C07308=1230.127,396.275,-78.801,-175.693,7.707,148.228
C07309=1230.123,396.522,-78.835,-175.692,7.710,148.228
C07310=1230.118,396.770,-78.868,-175.691,7.712,148.229
C07311=1230.115,397.018,-78.903,-175.691,7.714,148.229
C07312=1230.110,397.266,-78.936,-175.690,7.717,148.229
C07313=1230.106,397.513,-78.970,-175.689,7.719,148.230
C07314=1230.102,397.760,-79.004,-175.688,7.722,148.230
C07315=1230.098,398.009,-79.038,-175.688,7.724,148.231
C07316=1230.094,398.256,-79.072,-175.686,7.727,148.231
C07317=1230.090,398.503,-79.106,-175.686,7.729,148.232
C07318=1230.086,398.751,-79.141,-175.685,7.731,148.232
C07319=1230.082,398.999,-79.174,-175.684,7.734,148.232
C07320=1230.078,399.246,-79.208,-175.684,7.736,148.233
C07321=1230.073,399.494,-79.243,-175.683,7.739,148.233
C07322=1230.070,399.742,-79.276,-175.682,7.741,148.234
C07323=1230.065,399.989,-79.311,-175.681,7.743,148.234
C07324=1230.061,400.237,-79.345,-175.681,7.746,148.235
C07325=1230.057,400.485,-79.379,-175.680,7.748,148.235
C07326=1230.053,400.732,-79.413,-175.679,7.750,148.235
C07327=1230.049,400.980,-79.447,-175.678,7.753,148.236
C07328=1230.045,401.228,-79.481,-175.678,7.755,148.236
C07329=1230.041,401.475,-79.516,-175.677,7.758,148.237
C07330=1230.037,401.723,-79.549,-175.676,7.760,148.237
C07331=1230.033,401.971,-79.584,-175.676,7.762,148.237
C07332=1230.029,402.218,-79.618,-175.674,7.764,148.238
C07333=1230.024,402.465,-79.652,-175.674,7.767,148.238
C07334=1230.021,402.713,-79.686,-175.674,7.769,148.239
C07335=1230.016,402.961,-79.720,-175.672,7.772,148.239
C07336=1230.012,403.208,-79.754,-175.672,7.773,148.239
C07337=1230.008,403.456,-79.789,-175.672,7.776,148.240
C07338=1230.005,403.704,-79.823,-175.671,7.778,148.240
C07339=1230.000,403.951,-79.857,-175.670,7.781,148.241
C07340=1229.997,404.199,-79.891,-175.669,7.783,148.241
C07341=1229.992,404.446,-79.926,-175.669,7.785,148.241
C07342=1229.987,404.694,-79.960,-175.668,7.788,148.242
C07343=1229.984,404.942,-79.994,-175.667,7.790,148.242
C07344=1229.979,405.190,-80.028,-175.667,7.792,148.243
C07345=1229.976,405.437,-80.062,-175.666,7.795,148.243
C07346=1229.972,405.685,-80.097,-175.665,7.797,148.243
C07347=1229.968,405.932,-80.131,-175.665,7.799,148.244
C07348=1229.963,406.179,-80.165,-175.664,7.801,148.244
C07349=1229.960,406.427,-80.200,-175.663,7.804,148.245
C07350=1229.955,406.675,-80.233,-175.663,7.806,148.245
C07351=1229.951,406.923,-80.268,-175.662,7.808,148.245
C07352=1229.947,407.170,-80.302,-175.661,7.810,148.246
C07353=1229.943,407.418,-80.337,-175.661,7.813,148.246
C07354=1229.940,407.666,-80.371,-175.660,7.815,148.247
C07355=1229.935,407.913,-80.405,-175.659,7.817,148.247
C07356=1229.930,408.160,-80.440,-175.659,7.819,148.247
C07357=1229.927,408.408,-80.474,-175.658,7.822,148.248
C07358=1229.923,408.656,-80.508,-175.658,7.824,148.248
C07359=1229.919,408.904,-80.543,-175.657,7.826,148.249
C07360=1229.915,409.151,-80.577,-175.656,7.828,148.249
C07361=1229.910,409.398,-80.612,-175.656,7.831,148.250
C07362=1229.907,409.646,-80.646,-175.655,7.833,148.250
C07363=1229.902,409.894,-80.680,-175.654,7.835,148.250
C07364=1229.898,410.142,-80.715,-175.654,7.837,148.251
C07365=1229.895,410.389,-80.749,-175.653,7.839,148.251
C07366=1229.890,410.636,-80.783,-175.652,7.842,148.252
C07367=1229.886,410.884,-80.818,-175.652,7.844,148.252
C07368=1229.882,411.131,-80.852,-175.651,7.846,148.252
C07369=1229.878,411.380,-80.887,-175.651,7.848,148.253
C07370=1229.874,411.627,-80.921,-175.650,7.850,148.253
C07371=1229.870,411.874,-80.955,-175.650,7.852,148.254
C07372=1229.866,412.122,-80.990,-175.648,7.855,148.254
C07373=1229.861,412.370,-81.025,-175.648,7.857,148.254
C07374=1229.858,412.617,-81.059,-175.648,7.859,148.255
C07375=1229.854,412.865,-81.093,-175.647,7.861,148.255
C07376=1229.849,413.112,-81.128,-175.646,7.863,148.255
C07377=1229.846,413.360,-81.162,-175.646,7.865,148.256
C07378=1229.841,413.607,-81.196,-175.645,7.868,148.256
C07379=1229.837,413.856,-81.231,-175.644,7.870,148.257
C07380=1229.834,414.102,-81.266,-175.644,7.872,148.257
C07381=1229.830,414.350,-81.301,-175.644,7.875,148.258
C07382=1229.825,414.598,-81.335,-175.643,7.876,148.258
C07383=1229.822,414.845,-81.369,-175.642,7.878,148.258
C07384=1229.817,415.093,-81.404,-175.642,7.880,148.259
C07385=1229.813,415.340,-81.438,-175.641,7.884,148.259
C07386=1229.809,415.588,-81.473,-175.640,7.886,148.260
C07387=1229.803,415.965,-81.525,-175.640,7.889,148.260
C07388=1229.797,416.341,-81.578,-175.639,7.892,148.261
C07389=1229.791,416.718,-81.631,-175.638,7.895,148.261
C07390=1229.786,417.095,-81.684,-175.636,7.899,148.262
C07391=1229.363,417.096,-81.716,-175.640,7.909,148.266
C07392=1229.368,416.716,-81.663,-175.641,7.905,148.265
C07393=1229.374,416.336,-81.610,-175.642,7.902,148.264
C07394=1229.381,415.957,-81.557,-175.643,7.899,148.264
C07395=1229.387,415.578,-81.504,-175.643,7.896,148.263
C07396=1229.391,415.330,-81.470,-175.645,7.893,148.263
C07397=1229.395,415.082,-81.435,-175.645,7.891,148.262
C07398=1229.399,414.835,-81.401,-175.646,7.889,148.262
C07399=1229.403,414.587,-81.366,-175.646,7.887,148.262
C07400=1229.408,414.340,-81.332,-175.647,7.885,148.261
C07401=1229.411,414.092,-81.297,-175.647,7.883,148.261
C07402=1229.415,413.845,-81.262,-175.648,7.881,148.261
C07403=1229.419,413.597,-81.227,-175.648,7.879,148.260
C07404=1229.424,413.349,-81.193,-175.649,7.876,148.260
C07405=1229.428,413.102,-81.159,-175.650,7.874,148.259
C07406=1229.432,412.854,-81.124,-175.651,7.872,148.259
C07407=1229.436,412.607,-81.090,-175.651,7.870,148.258
C07408=1229.439,412.359,-81.056,-175.651,7.868,148.258
C07409=1229.444,412.112,-81.021,-175.652,7.866,148.258
C07410=1229.448,411.863,-80.986,-175.653,7.862,148.257
C07411=1229.452,411.616,-80.952,-175.653,7.861,148.257
C07412=1229.456,411.369,-80.918,-175.654,7.859,148.256
C07413=1229.460,411.121,-80.883,-175.655,7.857,148.256
C07414=1229.464,410.874,-80.849,-175.655,7.854,148.256
C07415=1229.468,410.626,-80.814,-175.656,7.851,148.255
C07416=1229.473,410.378,-80.780,-175.657,7.849,148.255
C07417=1229.477,410.131,-80.746,-175.657,7.847,148.254
C07418=1229.480,409.883,-80.711,-175.657,7.845,148.254
C07419=1229.485,409.635,-80.677,-175.658,7.843,148.254
C07420=1229.488,409.388,-80.643,-175.659,7.840,148.253
C07421=1229.493,409.140,-80.608,-175.660,7.838,148.253
C07422=1229.497,408.893,-80.574,-175.660,7.836,148.252
C07423=1229.501,408.645,-80.539,-175.661,7.834,148.252
C07424=1229.505,408.398,-80.505,-175.661,7.832,148.252
C07425=1229.508,408.150,-80.471,-175.662,7.829,148.251
C07426=1229.513,407.902,-80.436,-175.663,7.827,148.251
C07427=1229.518,407.655,-80.402,-175.663,7.825,148.250
C07428=1229.521,407.407,-80.367,-175.664,7.823,148.250
C07429=1229.525,407.160,-80.333,-175.665,7.820,148.249
C07430=1229.529,406.913,-80.299,-175.665,7.818,148.249
C07431=1229.533,406.665,-80.264,-175.666,7.816,148.249
C07432=1229.538,406.417,-80.230,-175.666,7.814,148.248
C07433=1229.541,406.169,-80.196,-175.667,7.811,148.248
C07434=1229.546,405.922,-80.161,-175.668,7.809,148.247
C07435=1229.550,405.674,-80.128,-175.668,7.807,148.247
C07436=1229.554,405.426,-80.093,-175.670,7.804,148.247
C07437=1229.558,405.179,-80.059,-175.670,7.802,148.246
C07438=1229.562,404.931,-80.025,-175.670,7.800,148.246
C07439=1229.566,404.683,-79.990,-175.671,7.798,148.245
C07440=1229.570,404.436,-79.956,-175.672,7.795,148.245
C07441=1229.574,404.189,-79.922,-175.672,7.793,148.244
C07442=1229.578,403.941,-79.887,-175.673,7.791,148.244
C07443=1229.583,403.693,-79.854,-175.674,7.788,148.244
C07444=1229.586,403.446,-79.820,-175.675,7.786,148.243
C07445=1229.590,403.198,-79.785,-175.675,7.784,148.243
C07446=1229.594,402.951,-79.751,-175.676,7.781,148.242
C07447=1229.598,402.703,-79.716,-175.677,7.779,148.242
C07448=1229.602,402.455,-79.682,-175.677,7.777,148.242
C07449=1229.607,402.207,-79.649,-175.678,7.774,148.241
C07450=1229.610,401.960,-79.614,-175.679,7.772,148.241
C07451=1229.615,401.712,-79.580,-175.679,7.770,148.240
C07452=1229.619,401.465,-79.545,-175.681,7.767,148.240
C07453=1229.623,401.218,-79.512,-175.681,7.765,148.240
C07454=1229.627,400.969,-79.477,-175.681,7.763,148.239
C07455=1229.631,400.722,-79.444,-175.683,7.760,148.239
C07456=1229.636,400.474,-79.409,-175.683,7.758,148.238
C07457=1229.639,400.227,-79.375,-175.684,7.756,148.238
C07458=1229.644,399.978,-79.341,-175.684,7.753,148.238
C07459=1229.648,399.731,-79.307,-175.685,7.751,148.237
C07460=1229.651,399.484,-79.273,-175.686,7.748,148.237
C07461=1229.655,399.236,-79.239,-175.687,7.746,148.236
C07462=1229.660,398.988,-79.205,-175.687,7.744,148.236
C07463=1229.664,398.740,-79.171,-175.688,7.741,148.235
C07464=1229.667,398.493,-79.137,-175.689,7.739,148.235
C07465=1229.672,398.245,-79.103,-175.690,7.736,148.235
C07466=1229.676,397.998,-79.069,-175.691,7.734,148.234
C07467=1229.680,397.750,-79.034,-175.691,7.732,148.234
C07468=1229.684,397.502,-79.001,-175.692,7.729,148.233
C07469=1229.689,397.255,-78.967,-175.693,7.727,148.233
C07470=1229.692,397.007,-78.932,-175.694,7.724,148.233
C07471=1229.696,396.759,-78.899,-175.694,7.722,148.232
C07472=1229.701,396.512,-78.865,-175.695,7.719,148.232
C07473=1229.705,396.265,-78.831,-175.696,7.717,148.231
C07474=1229.709,396.016,-78.797,-175.696,7.715,148.231
C07475=1229.713,395.769,-78.763,-175.698,7.713,148.231
C07476=1229.717,395.521,-78.728,-175.698,7.711,148.230
C07477=1229.721,395.274,-78.695,-175.699,7.707,148.230
C07478=1229.725,395.026,-78.661,-175.700,7.705,148.229
C07479=1229.729,394.778,-78.627,-175.701,7.703,148.229
C07480=1229.733,394.531,-78.593,-175.701,7.701,148.229
C07481=1229.738,394.283,-78.559,-175.702,7.698,148.228
C07482=1229.741,394.035,-78.525,-175.703,7.696,148.228
C07483=1229.745,393.788,-78.492,-175.704,7.693,148.227
C07484=1229.750,393.506,-78.453,-175.705,7.690,148.227
C07485=1229.755,393.225,-78.414,-175.706,7.688,148.227
C07486=1229.759,392.944,-78.375,-175.707,7.685,148.226
C07487=1229.764,392.662,-78.338,-175.708,7.682,148.226
C07488=1229.768,392.415,-78.304,-175.709,7.679,148.225
C07489=1229.773,392.167,-78.270,-175.709,7.677,148.225
C07490=1229.776,391.919,-78.236,-175.710,7.674,148.224
C07491=1229.780,391.672,-78.203,-175.711,7.672,148.224
C07492=1229.785,391.424,-78.168,-175.712,7.670,148.224
C07493=1229.789,391.176,-78.135,-175.712,7.667,148.223
C07494=1229.792,390.929,-78.101,-175.714,7.664,148.223
C07495=1229.797,390.681,-78.067,-175.715,7.662,148.222
C07496=1229.801,390.434,-78.033,-175.715,7.660,148.222
C07497=1229.805,390.186,-78.000,-175.717,7.657,148.222
C07498=1229.809,389.938,-77.965,-175.717,7.655,148.221
C07499=1229.813,389.690,-77.932,-175.718,7.652,148.221
C07500=1229.817,389.443,-77.898,-175.719,7.650,148.220
C07501=1229.821,389.195,-77.865,-175.720,7.647,148.220
C07502=1229.826,388.947,-77.831,-175.721,7.644,148.220
C07503=1229.829,388.699,-77.797,-175.722,7.642,148.219
C07504=1229.834,388.452,-77.764,-175.723,7.639,148.219
C07505=1229.838,388.204,-77.729,-175.723,7.637,148.218
C07506=1229.842,387.956,-77.696,-175.724,7.634,148.218
C07507=1229.846,387.709,-77.662,-175.726,7.632,148.218
C07508=1229.850,387.461,-77.629,-175.726,7.630,148.217
C07509=1229.855,387.213,-77.595,-175.727,7.627,148.217
C07510=1229.858,386.966,-77.561,-175.729,7.624,148.216
C07511=1229.862,386.718,-77.528,-175.729,7.622,148.216
C07512=1229.867,386.470,-77.495,-175.730,7.619,148.216
C07513=1229.871,386.223,-77.460,-175.732,7.616,148.215
C07514=1229.875,385.974,-77.427,-175.732,7.614,148.215
C07515=1229.879,385.727,-77.394,-175.733,7.612,148.215
C07516=1229.883,385.480,-77.360,-175.734,7.609,148.214
C07517=1229.887,385.232,-77.327,-175.735,7.607,148.214
C07518=1229.892,384.984,-77.293,-175.736,7.604,148.213
C07519=1229.896,384.737,-77.259,-175.737,7.601,148.213
C07520=1229.900,384.489,-77.226,-175.738,7.599,148.213
C07521=1229.903,384.241,-77.192,-175.739,7.596,148.212
C07522=1229.908,383.993,-77.158,-175.740,7.594,148.212
C07523=1229.912,383.745,-77.125,-175.741,7.592,148.212
C07524=1229.916,383.498,-77.092,-175.742,7.589,148.211
C07525=1229.920,383.250,-77.059,-175.743,7.586,148.211
C07526=1229.924,383.003,-77.025,-175.744,7.584,148.210
C07527=1229.928,382.755,-76.992,-175.745,7.581,148.210
C07528=1229.932,382.506,-76.957,-175.746,7.578,148.210
C07529=1229.937,382.259,-76.924,-175.747,7.575,148.209
C07530=1229.940,382.012,-76.890,-175.748,7.573,148.209
C07531=1229.945,381.764,-76.857,-175.749,7.571,148.208
C07532=1229.949,381.516,-76.824,-175.750,7.568,148.208
C07533=1229.953,381.268,-76.791,-175.752,7.565,148.208
C07534=1229.957,381.021,-76.758,-175.753,7.563,148.207
C07535=1229.962,380.773,-76.723,-175.754,7.560,148.207
C07536=1229.966,380.525,-76.690,-175.755,7.558,148.207
C07537=1229.970,380.278,-76.657,-175.756,7.555,148.206
C07538=1229.973,380.029,-76.623,-175.757,7.553,148.206
C07539=1229.978,379.782,-76.590,-175.758,7.550,148.206
C07540=1229.982,379.534,-76.557,-175.759,7.547,148.205
C07541=1229.985,379.287,-76.523,-175.760,7.544,148.205
C07542=1229.990,379.039,-76.490,-175.761,7.542,148.204
C07543=1229.994,378.791,-76.457,-175.763,7.540,148.204
C07544=1229.999,378.543,-76.423,-175.764,7.537,148.204
C07545=1230.003,378.295,-76.390,-175.765,7.534,148.203
C07546=1230.007,378.048,-76.357,-175.766,7.531,148.203
C07547=1230.011,377.800,-76.324,-175.767,7.529,148.203
C07548=1230.015,377.552,-76.291,-175.768,7.527,148.202
C07549=1230.019,377.305,-76.257,-175.769,7.524,148.202
C07550=1230.023,377.057,-76.224,-175.771,7.521,148.202
C07551=1230.028,376.809,-76.191,-175.772,7.518,148.201
C07552=1230.031,376.561,-76.158,-175.773,7.516,148.201
C07553=1230.035,376.314,-76.124,-175.774,7.513,148.200
C07554=1230.039,376.066,-76.091,-175.775,7.511,148.200
C07555=1230.043,375.818,-76.057,-175.776,7.508,148.200
C07556=1230.047,375.570,-76.024,-175.777,7.505,148.200
C07557=1230.052,375.323,-75.991,-175.779,7.503,148.199
C07558=1230.056,375.075,-75.958,-175.780,7.500,148.199
C07559=1230.060,374.827,-75.925,-175.781,7.497,148.199
C07560=1230.064,374.579,-75.892,-175.783,7.494,148.198
C07561=1230.068,374.331,-75.859,-175.784,7.492,148.198
C07562=1230.073,374.083,-75.826,-175.784,7.490,148.197
C07563=1230.077,373.836,-75.793,-175.786,7.487,148.197
C07564=1230.081,373.588,-75.760,-175.787,7.484,148.197
C07565=1230.085,373.340,-75.727,-175.788,7.481,148.196
C07566=1230.089,373.092,-75.693,-175.790,7.479,148.196
C07567=1230.093,372.845,-75.660,-175.791,7.476,148.196
C07568=1230.097,372.597,-75.627,-175.792,7.473,148.195
C07569=1230.101,372.349,-75.594,-175.793,7.470,148.195
C07570=1230.106,372.102,-75.561,-175.795,7.468,148.195
C07571=1230.110,371.854,-75.528,-175.796,7.465,148.194
C07572=1230.114,371.606,-75.494,-175.798,7.463,148.194
C07573=1230.118,371.358,-75.462,-175.799,7.460,148.194
C07574=1230.122,371.110,-75.429,-175.800,7.457,148.193
C07575=1230.126,370.863,-75.396,-175.801,7.455,148.193
C07576=1230.130,370.615,-75.363,-175.802,7.452,148.193
C07577=1230.134,370.367,-75.330,-175.804,7.450,148.193
C07578=1230.138,370.119,-75.297,-175.805,7.447,148.192
C07579=1230.143,369.871,-75.264,-175.806,7.444,148.192
C07580=1230.147,369.623,-75.231,-175.808,7.442,148.192
C07581=1230.151,369.376,-75.198,-175.809,7.439,148.191
C07582=1230.156,369.129,-75.165,-175.810,7.436,148.191
C07583=1230.160,368.881,-75.132,-175.812,7.433,148.191
C07584=1230.164,368.633,-75.100,-175.813,7.431,148.190
C07585=1230.168,368.385,-75.067,-175.815,7.428,148.190
C07586=1230.172,368.137,-75.034,-175.816,7.425,148.190
C07587=1230.176,367.890,-75.001,-175.818,7.423,148.190
C07588=1230.181,367.609,-74.964,-175.819,7.419,148.189
C07589=1230.185,367.330,-74.927,-175.820,7.416,148.189
C07590=1230.190,367.051,-74.891,-175.822,7.414,148.189
C07591=1230.195,366.771,-74.853,-175.824,7.410,148.188
C07592=1230.199,366.523,-74.820,-175.825,7.408,148.188
C07593=1230.202,366.276,-74.787,-175.826,7.405,148.188
C07594=1230.207,366.028,-74.755,-175.828,7.402,148.187
C07595=1230.211,365.780,-74.722,-175.829,7.399,148.187
C07596=1230.215,365.531,-74.689,-175.831,7.397,148.187
C07597=1230.220,365.284,-74.656,-175.832,7.394,148.186
C07598=1230.224,365.037,-74.624,-175.834,7.391,148.186
C07599=1230.228,364.789,-74.592,-175.835,7.389,148.186
C07600=1230.232,364.541,-74.558,-175.836,7.386,148.186
C07601=1230.236,364.293,-74.525,-175.838,7.384,148.185
C07602=1230.240,364.045,-74.493,-175.839,7.381,148.185
C07603=1230.244,363.797,-74.460,-175.841,7.378,148.185
C07604=1230.249,363.549,-74.428,-175.842,7.375,148.184
C07605=1230.253,363.301,-74.395,-175.844,7.373,148.184
C07606=1230.256,363.053,-74.363,-175.845,7.370,148.184
C07607=1230.261,362.806,-74.330,-175.847,7.367,148.184
C07608=1230.265,362.559,-74.297,-175.849,7.364,148.183
C07609=1230.269,362.311,-74.265,-175.850,7.361,148.183
C07610=1230.273,362.063,-74.232,-175.851,7.359,148.183
C07611=1230.278,361.814,-74.199,-175.853,7.356,148.183
C07612=1230.281,361.567,-74.167,-175.854,7.353,148.182
C07613=1230.285,361.319,-74.134,-175.856,7.351,148.182
C07614=1230.290,361.072,-74.102,-175.857,7.348,148.182
C07615=1230.294,360.824,-74.070,-175.859,7.346,148.181
C07616=1230.298,360.575,-74.037,-175.860,7.343,148.181
C07617=1230.302,360.328,-74.004,-175.862,7.340,148.181
C07618=1230.306,360.080,-73.972,-175.864,7.337,148.181
C07619=1230.310,359.832,-73.939,-175.865,7.334,148.180
C07620=1230.315,359.584,-73.907,-175.867,7.332,148.180
C07621=1230.319,359.337,-73.875,-175.868,7.329,148.180
C07622=1230.323,359.088,-73.842,-175.870,7.327,148.180
C07623=1230.328,358.840,-73.810,-175.871,7.324,148.179
C07624=1230.331,358.593,-73.777,-175.873,7.321,148.179
C07625=1230.336,358.345,-73.745,-175.874,7.319,148.179
C07626=1230.339,358.098,-73.712,-175.877,7.315,148.179
C07627=1230.344,357.849,-73.680,-175.878,7.313,148.178
C07628=1230.348,357.601,-73.648,-175.879,7.310,148.178
C07629=1230.352,357.353,-73.615,-175.881,7.308,148.178
C07630=1230.357,357.106,-73.583,-175.883,7.305,148.178
C07631=1230.361,356.858,-73.551,-175.884,7.302,148.178
C07632=1230.365,356.609,-73.519,-175.885,7.300,148.177
C07633=1230.368,356.362,-73.486,-175.887,7.297,148.177
C07634=1230.373,356.114,-73.454,-175.889,7.294,148.177
C07635=1230.378,355.866,-73.422,-175.891,7.291,148.177
C07636=1230.381,355.619,-73.389,-175.892,7.289,148.177
C07637=1230.386,355.370,-73.357,-175.894,7.286,148.176
C07638=1230.390,355.123,-73.325,-175.895,7.283,148.176
C07639=1230.394,354.875,-73.293,-175.897,7.281,148.176
C07640=1230.398,354.627,-73.260,-175.899,7.277,148.176
C07641=1230.402,354.379,-73.228,-175.901,7.275,148.175
C07642=1230.407,354.131,-73.196,-175.902,7.272,148.175
C07643=1230.411,353.883,-73.164,-175.904,7.270,148.175
C07644=1230.415,353.635,-73.132,-175.906,7.267,148.175
C07645=1230.419,353.387,-73.099,-175.907,7.265,148.175
C07646=1230.423,353.140,-73.067,-175.909,7.261,148.174
C07647=1230.428,352.892,-73.035,-175.911,7.259,148.174
C07648=1230.431,352.644,-73.003,-175.912,7.256,148.174
C07649=1230.436,352.396,-72.971,-175.914,7.253,148.174
C07650=1230.440,352.148,-72.939,-175.915,7.251,148.173
C07651=1230.445,351.900,-72.907,-175.917,7.248,148.173
C07652=1230.448,351.651,-72.875,-175.919,7.245,148.173
C07653=1230.452,351.405,-72.843,-175.921,7.243,148.173
C07654=1230.457,351.156,-72.810,-175.922,7.240,148.173
C07655=1230.460,350.908,-72.778,-175.924,7.237,148.172
C07656=1230.465,350.661,-72.746,-175.926,7.235,148.172
C07657=1230.469,350.413,-72.714,-175.927,7.232,148.172
C07658=1230.473,350.165,-72.683,-175.929,7.229,148.172
C07659=1230.478,349.917,-72.650,-175.931,7.226,148.172
C07660=1230.482,349.669,-72.619,-175.933,7.224,148.172
C07661=1230.486,349.421,-72.586,-175.934,7.221,148.171
C07662=1230.490,349.173,-72.555,-175.936,7.219,148.171
C07663=1230.494,348.925,-72.523,-175.938,7.216,148.171
C07664=1230.499,348.677,-72.490,-175.940,7.213,148.171
C07665=1230.503,348.430,-72.459,-175.941,7.210,148.171
C07666=1230.507,348.182,-72.427,-175.943,7.208,148.171
C07667=1230.511,347.933,-72.395,-175.945,7.206,148.170
C07668=1230.515,347.686,-72.363,-175.947,7.202,148.170
C07669=1230.519,347.438,-72.331,-175.949,7.200,148.170
C07670=1230.524,347.190,-72.300,-175.951,7.197,148.170
C07671=1230.528,346.941,-72.268,-175.952,7.195,148.170
C07672=1230.532,346.693,-72.236,-175.954,7.191,148.169
C07673=1230.537,346.446,-72.204,-175.956,7.189,148.169
C07674=1230.541,346.198,-72.172,-175.958,7.186,148.169
C07675=1230.545,345.950,-72.141,-175.959,7.184,148.169
C07676=1230.549,345.702,-72.108,-175.961,7.182,148.169
C07677=1230.553,345.454,-72.077,-175.963,7.178,148.169
C07678=1230.558,345.206,-72.046,-175.965,7.176,148.168
C07679=1230.561,344.958,-72.014,-175.967,7.173,148.168
C07680=1230.566,344.710,-71.982,-175.968,7.171,148.168
C07681=1230.570,344.462,-71.950,-175.970,7.167,148.168
C07682=1230.574,344.214,-71.918,-175.973,7.165,148.168
C07683=1230.578,343.966,-71.887,-175.974,7.162,148.168
C07684=1230.583,343.718,-71.855,-175.976,7.160,148.168
C07685=1230.587,343.471,-71.824,-175.977,7.157,148.167
C07686=1230.591,343.223,-71.792,-175.980,7.154,148.167
C07687=1230.595,342.975,-71.761,-175.982,7.152,148.167
C07688=1230.600,342.726,-71.728,-175.983,7.149,148.167
C07689=1230.604,342.478,-71.697,-175.985,7.147,148.167
C07690=1230.608,342.231,-71.665,-175.987,7.143,148.167
C07691=1230.612,341.982,-71.634,-175.989,7.141,148.167
C07692=1230.617,341.705,-71.599,-175.991,7.139,148.166
C07693=1230.621,341.428,-71.563,-175.993,7.135,148.166
C07694=1230.626,341.149,-71.528,-175.995,7.132,148.166
C07695=1230.631,340.873,-71.492,-175.997,7.130,148.166
C07696=1230.635,340.624,-71.461,-175.999,7.126,148.166
C07697=1230.640,340.377,-71.430,-176.001,7.124,148.166
C07698=1230.643,340.129,-71.398,-176.003,7.121,148.166
C07699=1230.648,339.881,-71.367,-176.005,7.119,148.165
C07700=1230.652,339.633,-71.335,-176.007,7.116,148.165
C07701=1230.656,339.385,-71.305,-176.009,7.113,148.165
C07702=1230.661,339.136,-71.272,-176.011,7.111,148.165
C07703=1230.665,338.889,-71.241,-176.012,7.108,148.165
C07704=1230.669,338.640,-71.210,-176.014,7.105,148.165
C07705=1230.673,338.393,-71.178,-176.017,7.103,148.165
C07706=1230.677,338.144,-71.147,-176.018,7.100,148.164
C07707=1230.682,337.897,-71.115,-176.020,7.098,148.164
C07708=1230.686,337.648,-71.084,-176.022,7.095,148.164
C07709=1230.690,337.401,-71.053,-176.024,7.092,148.164
C07710=1230.694,337.152,-71.022,-176.026,7.090,148.164
C07711=1230.698,336.905,-70.990,-176.028,7.087,148.164
C07712=1230.702,336.656,-70.959,-176.030,7.084,148.164
C07713=1230.707,336.409,-70.928,-176.032,7.082,148.164
C07714=1230.711,336.160,-70.897,-176.034,7.079,148.164
C07715=1230.715,335.913,-70.865,-176.036,7.077,148.164
C07716=1230.719,335.664,-70.834,-176.038,7.074,148.163
C07717=1230.724,335.416,-70.803,-176.040,7.071,148.163
C07718=1230.728,335.169,-70.772,-176.042,7.069,148.163
C07719=1230.732,334.920,-70.741,-176.043,7.066,148.163
C07720=1230.736,334.673,-70.709,-176.046,7.063,148.163
C07721=1230.740,334.424,-70.678,-176.048,7.061,148.163
C07722=1230.745,334.176,-70.647,-176.049,7.058,148.163
C07723=1230.749,333.928,-70.615,-176.051,7.056,148.163
C07724=1230.753,333.680,-70.585,-176.053,7.053,148.163
C07725=1230.758,333.432,-70.554,-176.056,7.050,148.163
C07726=1230.762,333.184,-70.522,-176.057,7.048,148.162
C07727=1230.766,332.936,-70.491,-176.060,7.045,148.162
C07728=1230.770,332.688,-70.460,-176.061,7.042,148.162
C07729=1230.774,332.440,-70.429,-176.064,7.040,148.162
C07730=1230.779,332.193,-70.398,-176.065,7.037,148.162
C07731=1230.783,331.944,-70.367,-176.068,7.034,148.162
C07732=1230.787,331.696,-70.337,-176.069,7.032,148.162
C07733=1230.791,331.449,-70.305,-176.072,7.030,148.162
C07734=1230.795,331.200,-70.274,-176.073,7.027,148.162
C07735=1230.800,330.952,-70.243,-176.076,7.024,148.162
C07736=1230.804,330.704,-70.212,-176.077,7.021,148.162
C07737=1230.809,330.456,-70.181,-176.080,7.019,148.162
C07738=1230.813,330.208,-70.150,-176.082,7.016,148.161
C07739=1230.817,329.960,-70.119,-176.084,7.014,148.161
C07740=1230.821,329.712,-70.088,-176.086,7.011,148.161
C07741=1230.825,329.464,-70.058,-176.088,7.009,148.161
C07742=1230.829,329.215,-70.027,-176.090,7.006,148.161
C07743=1230.834,328.967,-69.996,-176.092,7.003,148.161
C07744=1230.838,328.720,-69.964,-176.094,7.001,148.161
C07745=1230.842,328.472,-69.934,-176.095,6.999,148.161
C07746=1230.846,328.224,-69.903,-176.098,6.995,148.161
C07747=1230.851,327.976,-69.872,-176.100,6.993,148.161
C07748=1230.855,327.727,-69.841,-176.102,6.991,148.161
C07749=1230.859,327.479,-69.810,-176.104,6.988,148.161
C07750=1230.863,327.232,-69.780,-176.106,6.985,148.161
C07751=1230.868,326.984,-69.749,-176.108,6.983,148.161
C07752=1230.872,326.735,-69.718,-176.110,6.981,148.161
C07753=1230.877,326.487,-69.688,-176.112,6.977,148.160
C07754=1230.880,326.239,-69.657,-176.115,6.975,148.161
C07755=1230.884,325.991,-69.626,-176.117,6.973,148.161
C07756=1230.889,325.743,-69.596,-176.118,6.970,148.160
C07757=1230.894,325.495,-69.565,-176.121,6.967,148.160
C07758=1230.898,325.247,-69.535,-176.123,6.965,148.160
C07759=1230.902,324.998,-69.503,-176.125,6.962,148.160
C07760=1230.906,324.750,-69.473,-176.127,6.959,148.160
C07761=1230.910,324.503,-69.443,-176.129,6.957,148.160
C07762=1230.914,324.254,-69.411,-176.131,6.955,148.160
C07763=1230.919,324.006,-69.381,-176.133,6.952,148.160
C07764=1230.923,323.759,-69.350,-176.136,6.949,148.160
C07765=1230.927,323.511,-69.320,-176.137,6.947,148.160
C07766=1230.932,323.263,-69.289,-176.140,6.945,148.160
C07767=1230.935,323.014,-69.259,-176.142,6.941,148.160
C07768=1230.940,322.766,-69.228,-176.144,6.939,148.160
C07769=1230.945,322.518,-69.198,-176.146,6.937,148.160
C07770=1230.948,322.270,-69.167,-176.148,6.935,148.160
C07771=1230.952,322.021,-69.136,-176.151,6.931,148.160
C07772=1230.956,321.774,-69.106,-176.153,6.929,148.160
C07773=1230.961,321.525,-69.076,-176.154,6.927,148.160
C07774=1230.966,321.277,-69.045,-176.156,6.924,148.160
C07775=1230.970,321.030,-69.015,-176.159,6.921,148.160
C07776=1230.974,320.781,-68.984,-176.161,6.919,148.160
C07777=1230.978,320.533,-68.954,-176.163,6.917,148.160
C07778=1230.983,320.285,-68.924,-176.165,6.914,148.160
C07779=1230.987,320.037,-68.893,-176.168,6.911,148.160
C07780=1230.991,319.789,-68.863,-176.170,6.909,148.160
C07781=1230.995,319.540,-68.832,-176.171,6.907,148.160
C07782=1230.999,319.292,-68.802,-176.174,6.904,148.160
C07783=1231.004,319.044,-68.771,-176.176,6.901,148.160
C07784=1231.008,318.797,-68.741,-176.178,6.899,148.160
C07785=1231.013,318.548,-68.711,-176.181,6.896,148.160
C07786=1231.017,318.300,-68.681,-176.182,6.893,148.160
C07787=1231.021,318.052,-68.650,-176.184,6.891,148.160
C07788=1231.025,317.803,-68.621,-176.187,6.889,148.160
C07789=1231.029,317.556,-68.590,-176.189,6.886,148.160
C07790=1231.033,317.307,-68.560,-176.191,6.884,148.160
C07791=1231.038,317.059,-68.530,-176.193,6.882,148.160
C07792=1231.042,316.812,-68.499,-176.195,6.879,148.160
C07793=1231.047,316.563,-68.469,-176.198,6.876,148.160
C07794=1231.051,316.315,-68.439,-176.200,6.874,148.160
C07795=1231.055,316.066,-68.409,-176.202,6.871,148.160
C07796=1231.060,315.791,-68.375,-176.205,6.868,148.160
C07797=1231.065,315.515,-68.342,-176.207,6.865,148.160
C07798=1231.069,315.239,-68.308,-176.209,6.863,148.160
C07799=1231.074,314.964,-68.276,-176.212,6.860,148.160
C07800=1231.078,314.716,-68.245,-176.214,6.858,148.160
C07801=1231.083,314.468,-68.215,-176.216,6.856,148.160
C07802=1231.087,314.220,-68.185,-176.219,6.853,148.160
C07803=1231.091,313.971,-68.155,-176.221,6.850,148.160
C07804=1231.095,313.723,-68.125,-176.223,6.848,148.160
C07805=1231.100,313.475,-68.095,-176.225,6.846,148.160
C07806=1231.103,313.227,-68.064,-176.227,6.842,148.160
C07807=1231.108,312.978,-68.034,-176.229,6.840,148.160
C07808=1231.113,312.730,-68.005,-176.231,6.838,148.160
C07809=1231.116,312.483,-67.975,-176.234,6.835,148.160
C07810=1231.121,312.234,-67.945,-176.236,6.833,148.160
C07811=1231.125,311.986,-67.915,-176.238,6.831,148.160
C07812=1231.129,311.738,-67.885,-176.240,6.828,148.160
C07813=1231.134,311.490,-67.855,-176.243,6.825,148.160
C07814=1231.138,311.242,-67.825,-176.245,6.823,148.160
C07815=1231.142,310.994,-67.795,-176.247,6.821,148.160
C07816=1231.147,310.745,-67.766,-176.249,6.819,148.160
C07817=1231.151,310.497,-67.735,-176.252,6.815,148.160
C07818=1231.155,310.249,-67.706,-176.254,6.813,148.160
C07819=1231.160,310.001,-67.676,-176.256,6.811,148.160
C07820=1231.164,309.752,-67.646,-176.258,6.809,148.160
C07821=1231.168,309.505,-67.616,-176.261,6.806,148.160
C07822=1231.173,309.256,-67.587,-176.263,6.804,148.160
C07823=1231.177,309.008,-67.557,-176.265,6.801,148.160
C07824=1231.182,308.759,-67.527,-176.268,6.798,148.160
C07825=1231.186,308.512,-67.497,-176.270,6.796,148.160
C07826=1231.190,308.264,-67.467,-176.272,6.794,148.160
C07827=1231.194,308.015,-67.438,-176.274,6.792,148.160
C07828=1231.198,307.767,-67.409,-176.277,6.789,148.160
C07829=1231.203,307.518,-67.379,-176.279,6.786,148.161
C07830=1231.207,307.271,-67.348,-176.281,6.784,148.161
C07831=1231.211,307.023,-67.319,-176.283,6.782,148.161
C07832=1231.215,306.774,-67.289,-176.286,6.779,148.161
C07833=1231.219,306.526,-67.260,-176.288,6.777,148.161
C07834=1231.224,306.277,-67.230,-176.290,6.774,148.161
C07835=1231.228,306.029,-67.200,-176.292,6.772,148.161
C07836=1231.233,305.781,-67.171,-176.295,6.769,148.161
C07837=1231.237,305.533,-67.142,-176.297,6.767,148.161
C07838=1231.242,305.285,-67.112,-176.299,6.765,148.161
C07839=1231.246,305.037,-67.082,-176.301,6.762,148.161
C07840=1231.250,304.789,-67.053,-176.304,6.760,148.161
C07841=1231.255,304.541,-67.023,-176.306,6.757,148.161
C07842=1231.259,304.292,-66.993,-176.308,6.755,148.161
C07843=1231.263,304.044,-66.964,-176.310,6.753,148.161
C07844=1231.267,303.796,-66.934,-176.313,6.750,148.161
C07845=1231.271,303.548,-66.905,-176.315,6.748,148.161
C07846=1231.276,303.299,-66.876,-176.317,6.745,148.161
C07847=1231.280,303.052,-66.846,-176.319,6.743,148.162
C07848=1231.284,302.803,-66.817,-176.322,6.740,148.162
C07849=1231.289,302.555,-66.788,-176.325,6.738,148.162
C07850=1231.293,302.306,-66.759,-176.327,6.736,148.162
C07851=1231.297,302.058,-66.729,-176.329,6.734,148.162
C07852=1231.302,301.810,-66.700,-176.331,6.731,148.162
C07853=1231.306,301.561,-66.670,-176.334,6.729,148.162
C07854=1231.310,301.313,-66.641,-176.336,6.726,148.162
C07855=1231.315,301.066,-66.612,-176.338,6.724,148.162
C07856=1231.319,300.817,-66.582,-176.340,6.722,148.162
C07857=1231.323,300.569,-66.553,-176.343,6.719,148.162
C07858=1231.327,300.321,-66.524,-176.345,6.717,148.162
C07859=1231.332,300.072,-66.495,-176.347,6.715,148.162
C07860=1231.336,299.824,-66.465,-176.349,6.712,148.163
C07861=1231.341,299.576,-66.436,-176.352,6.709,148.163
C07862=1231.345,299.328,-66.407,-176.355,6.707,148.163
C07863=1231.349,299.080,-66.377,-176.357,6.705,148.163
C07864=1231.354,298.831,-66.349,-176.359,6.703,148.163
C07865=1231.358,298.582,-66.319,-176.361,6.700,148.163
C07866=1231.362,298.335,-66.290,-176.364,6.698,148.163
C07867=1231.367,298.087,-66.261,-176.366,6.696,148.163
C07868=1231.371,297.838,-66.232,-176.368,6.694,148.163
C07869=1231.375,297.589,-66.202,-176.370,6.691,148.163
C07870=1231.380,297.341,-66.173,-176.373,6.688,148.163
C07871=1231.384,297.094,-66.144,-176.375,6.686,148.163
C07872=1231.389,296.845,-66.115,-176.378,6.684,148.164
C07873=1231.392,296.597,-66.086,-176.380,6.682,148.164
C07874=1231.396,296.348,-66.057,-176.382,6.679,148.164
C07875=1231.401,296.100,-66.028,-176.385,6.677,148.164
C07876=1231.406,295.852,-65.999,-176.387,6.674,148.164
C07877=1231.410,295.604,-65.970,-176.389,6.673,148.164
C07878=1231.414,295.355,-65.941,-176.391,6.670,148.164
C07879=1231.418,295.107,-65.912,-176.394,6.667,148.164
C07880=1231.423,294.859,-65.884,-176.396,6.665,148.164
C07881=1231.427,294.610,-65.854,-176.399,6.663,148.165
C07882=1231.431,294.362,-65.825,-176.401,6.661,148.165
C07883=1231.436,294.113,-65.796,-176.403,6.658,148.165
C07884=1231.441,293.866,-65.767,-176.406,6.656,148.165
C07885=1231.444,293.617,-65.739,-176.408,6.654,148.165
C07886=1231.448,293.369,-65.709,-176.410,6.652,148.165
C07887=1231.454,293.121,-65.681,-176.412,6.649,148.165
C07888=1231.458,292.872,-65.651,-176.416,6.647,148.165
C07889=1231.461,292.624,-65.623,-176.418,6.644,148.165
C07890=1231.466,292.376,-65.594,-176.420,6.642,148.165
C07891=1231.471,292.127,-65.565,-176.422,6.640,148.166
C07892=1231.475,291.879,-65.536,-176.424,6.638,148.166
C07893=1231.479,291.631,-65.508,-176.427,6.635,148.166
C07894=1231.483,291.383,-65.479,-176.429,6.633,148.166
C07895=1231.488,291.134,-65.450,-176.432,6.631,148.166
C07896=1231.492,290.886,-65.421,-176.434,6.629,148.166
C07897=1231.496,290.638,-65.393,-176.436,6.626,148.166
C07898=1231.501,290.389,-65.364,-176.439,6.624,148.167
C07899=1231.505,290.141,-65.335,-176.441,6.621,148.167
C07900=1231.511,289.867,-65.303,-176.443,6.619,148.167
C07901=1231.515,289.593,-65.272,-176.446,6.616,148.167
C07902=1231.519,289.319,-65.241,-176.449,6.614,148.167
C07903=1231.524,289.044,-65.209,-176.452,6.611,148.167
C07904=1231.529,288.797,-65.180,-176.454,6.609,148.167
C07905=1231.533,288.548,-65.152,-176.456,6.607,148.168
C07906=1231.537,288.299,-65.123,-176.459,6.605,148.168
C07907=1231.542,288.052,-65.094,-176.461,6.602,148.168
C07908=1231.546,287.803,-65.066,-176.464,6.600,148.168
C07909=1231.551,287.555,-65.037,-176.466,6.598,148.168
C07910=1231.555,287.307,-65.008,-176.468,6.596,148.168
C07911=1231.559,287.058,-64.980,-176.471,6.594,148.168
C07912=1231.564,286.810,-64.952,-176.473,6.591,148.168
C07913=1231.568,286.561,-64.923,-176.476,6.589,148.169
C07914=1231.573,286.313,-64.895,-176.478,6.587,148.169
C07915=1231.577,286.065,-64.866,-176.480,6.584,148.169
C07916=1231.581,285.816,-64.837,-176.483,6.583,148.169
C07917=1231.586,285.568,-64.809,-176.485,6.580,148.169
C07918=1231.589,285.320,-64.781,-176.487,6.577,148.169
C07919=1231.595,285.071,-64.753,-176.490,6.575,148.169
C07920=1231.598,284.823,-64.724,-176.492,6.573,148.169
C07921=1231.603,284.575,-64.695,-176.495,6.571,148.170
C07922=1231.607,284.327,-64.667,-176.497,6.569,148.170
C07923=1231.612,284.079,-64.639,-176.499,6.567,148.170
C07924=1231.616,283.830,-64.611,-176.502,6.564,148.170
C07925=1231.620,283.581,-64.582,-176.504,6.562,148.170
C07926=1231.625,283.333,-64.554,-176.507,6.560,148.170
C07927=1231.629,283.084,-64.525,-176.509,6.558,148.171
C07928=1231.633,282.836,-64.498,-176.511,6.556,148.171
C07929=1231.638,282.588,-64.469,-176.514,6.554,148.171
C07930=1231.642,282.340,-64.441,-176.516,6.551,148.171
C07931=1231.647,282.091,-64.412,-176.519,6.549,148.171
C07932=1231.651,281.843,-64.385,-176.521,6.546,148.171
C07933=1231.656,281.594,-64.356,-176.523,6.544,148.172
C07934=1231.660,281.346,-64.328,-176.526,6.542,148.172
C07935=1231.664,281.098,-64.300,-176.528,6.540,148.172
C07936=1231.669,280.849,-64.272,-176.530,6.538,148.172
C07937=1231.672,280.601,-64.243,-176.533,6.535,148.172
C07938=1231.678,280.353,-64.215,-176.536,6.533,148.172
C07939=1231.681,280.104,-64.187,-176.538,6.531,148.173
C07940=1231.686,279.856,-64.159,-176.540,6.529,148.173
C07941=1231.690,279.607,-64.130,-176.543,6.527,148.173
C07942=1231.694,279.359,-64.103,-176.545,6.525,148.173
C07943=1231.698,279.111,-64.074,-176.547,6.523,148.173
C07944=1231.703,278.863,-64.046,-176.550,6.520,148.173
C07945=1231.708,278.615,-64.018,-176.552,6.518,148.173
C07946=1231.712,278.366,-63.991,-176.555,6.516,148.174
C07947=1231.717,278.117,-63.962,-176.557,6.514,148.174
C07948=1231.721,277.869,-63.934,-176.560,6.512,148.174
C07949=1231.725,277.621,-63.907,-176.562,6.510,148.174
C07950=1231.729,277.372,-63.878,-176.564,6.508,148.174
C07951=1231.734,277.124,-63.850,-176.566,6.505,148.174
C07952=1231.738,276.875,-63.823,-176.570,6.503,148.175
C07953=1231.743,276.627,-63.794,-176.572,6.500,148.175
C07954=1231.747,276.379,-63.766,-176.574,6.499,148.175
C07955=1231.751,276.130,-63.738,-176.576,6.496,148.175
C07956=1231.756,275.882,-63.711,-176.579,6.494,148.175
C07957=1231.760,275.633,-63.683,-176.582,6.493,148.176
C07958=1231.765,275.385,-63.655,-176.584,6.490,148.176
C07959=1231.769,275.137,-63.627,-176.586,6.488,148.176
C07960=1231.773,274.888,-63.600,-176.589,6.485,148.176
C07961=1231.778,274.640,-63.571,-176.592,6.483,148.176
C07962=1231.782,274.391,-63.543,-176.594,6.481,148.176
C07963=1231.786,274.143,-63.516,-176.596,6.479,148.177
C07964=1231.791,273.895,-63.488,-176.598,6.477,148.177
C07965=1231.795,273.646,-63.459,-176.601,6.475,148.177
C07966=1231.800,273.397,-63.432,-176.603,6.473,148.177
C07967=1231.804,273.150,-63.405,-176.606,6.471,148.177
C07968=1231.808,272.900,-63.377,-176.608,6.469,148.178
C07969=1231.813,272.653,-63.349,-176.611,6.466,148.178
C07970=1231.817,272.405,-63.322,-176.614,6.464,148.178
C07971=1231.822,272.155,-63.294,-176.616,6.462,148.178
C07972=1231.826,271.907,-63.266,-176.618,6.460,148.178
C07973=1231.831,271.659,-63.239,-176.620,6.458,148.178
C07974=1231.835,271.410,-63.211,-176.623,6.456,148.179
C07975=1231.839,271.162,-63.184,-176.625,6.454,148.179
C07976=1231.844,270.914,-63.156,-176.628,6.452,148.179
C07977=1231.848,270.665,-63.128,-176.630,6.450,148.179
C07978=1231.853,270.416,-63.100,-176.632,6.448,148.180
C07979=1231.857,270.168,-63.073,-176.635,6.446,148.180
C07980=1231.861,269.919,-63.045,-176.638,6.443,148.180
C07981=1231.866,269.671,-63.018,-176.640,6.441,148.180
C07982=1231.870,269.423,-62.990,-176.643,6.439,148.180
C07983=1231.875,269.175,-62.963,-176.645,6.437,148.181
C07984=1231.879,268.926,-62.935,-176.648,6.435,148.181
C07985=1231.883,268.677,-62.908,-176.650,6.433,148.181
C07986=1231.888,268.429,-62.881,-176.652,6.431,148.181
C07987=1231.892,268.181,-62.853,-176.655,6.429,148.181
C07988=1231.896,267.932,-62.825,-176.657,6.427,148.182
C07989=1231.901,267.684,-62.798,-176.660,6.425,148.182
C07990=1231.905,267.436,-62.771,-176.662,6.423,148.182
C07991=1231.909,267.186,-62.743,-176.664,6.421,148.182
C07992=1231.914,266.938,-62.715,-176.667,6.418,148.182
C07993=1231.918,266.690,-62.688,-176.670,6.416,148.183
C07994=1231.923,266.441,-62.661,-176.672,6.414,148.183
C07995=1231.927,266.194,-62.633,-176.675,6.412,148.183
C07996=1231.931,265.944,-62.606,-176.677,6.410,148.183
C07997=1231.936,265.696,-62.579,-176.680,6.408,148.184
C07998=1231.940,265.448,-62.551,-176.682,6.406,148.184
C07999=1231.945,265.200,-62.524,-176.684,6.404,148.184
C08000=1231.949,264.950,-62.497,-176.687,6.402,148.184
C08001=1231.954,264.702,-62.470,-176.689,6.400,148.184
C08002=1231.958,264.454,-62.442,-176.692,6.398,148.185
C08003=1231.963,264.205,-62.415,-176.694,6.396,148.185
C08004=1231.967,263.933,-62.385,-176.697,6.393,148.185
C08005=1231.973,263.660,-62.356,-176.699,6.391,148.185
C08006=1231.977,263.388,-62.326,-176.702,6.389,148.185
C08007=1231.983,263.115,-62.295,-176.705,6.386,148.186
C08008=1231.986,262.866,-62.269,-176.708,6.384,148.186
C08009=1231.991,262.618,-62.242,-176.710,6.382,148.186
C08010=1231.995,262.369,-62.215,-176.712,6.380,148.186
C08011=1232.000,262.121,-62.187,-176.715,6.378,148.187
C08012=1232.004,261.873,-62.160,-176.717,6.376,148.187
C08013=1232.009,261.624,-62.133,-176.720,6.374,148.187
C08014=1232.013,261.375,-62.105,-176.722,6.372,148.187
C08015=1232.017,261.127,-62.079,-176.725,6.370,148.187
C08016=1232.022,260.878,-62.052,-176.727,6.368,148.188
C08017=1232.026,260.630,-62.025,-176.730,6.366,148.188
C08018=1232.031,260.381,-61.998,-176.732,6.364,148.188
C08019=1232.036,260.133,-61.970,-176.734,6.362,148.188
C08020=1232.040,259.884,-61.943,-176.737,6.360,148.189
C08021=1232.044,259.636,-61.917,-176.739,6.358,148.189
C08022=1232.048,259.387,-61.890,-176.742,6.356,148.189
C08023=1232.053,259.138,-61.862,-176.744,6.354,148.189
C08024=1232.057,258.890,-61.835,-176.747,6.353,148.190
C08025=1232.061,258.642,-61.809,-176.749,6.350,148.190
C08026=1232.066,258.393,-61.782,-176.752,6.348,148.190
C08027=1232.071,258.145,-61.755,-176.754,6.347,148.190
C08028=1232.075,257.896,-61.728,-176.756,6.344,148.191
C08029=1232.079,257.648,-61.701,-176.759,6.342,148.191
C08030=1232.084,257.400,-61.674,-176.762,6.341,148.191
C08031=1232.089,257.151,-61.647,-176.764,6.339,148.191
C08032=1232.093,256.903,-61.620,-176.766,6.336,148.191
C08033=1232.097,256.654,-61.594,-176.769,6.335,148.192
C08034=1232.101,256.405,-61.566,-176.772,6.333,148.192
C08035=1232.106,256.156,-61.540,-176.774,6.330,148.192
C08036=1232.110,255.908,-61.513,-176.776,6.329,148.192
C08037=1232.115,255.659,-61.486,-176.779,6.327,148.193
C08038=1232.119,255.411,-61.459,-176.782,6.325,148.193
C08039=1232.123,255.163,-61.433,-176.784,6.323,148.193
C08040=1232.128,254.914,-61.406,-176.786,6.321,148.193
C08041=1232.133,254.665,-61.379,-176.789,6.319,148.194
C08042=1232.137,254.417,-61.353,-176.791,6.317,148.194
C08043=1232.142,254.168,-61.326,-176.794,6.315,148.194
C08044=1232.146,253.920,-61.299,-176.796,6.313,148.194
C08045=1232.150,253.671,-61.273,-176.799,6.311,148.195
C08046=1232.155,253.423,-61.246,-176.801,6.309,148.195
C08047=1232.159,253.175,-61.220,-176.804,6.307,148.195
C08048=1232.164,252.926,-61.192,-176.806,6.305,148.195
C08049=1232.169,252.677,-61.166,-176.809,6.303,148.196
C08050=1232.173,252.429,-61.140,-176.811,6.301,148.196
C08051=1232.177,252.180,-61.113,-176.813,6.299,148.196
C08052=1232.181,251.931,-61.087,-176.816,6.297,148.196
C08053=1232.186,251.683,-61.060,-176.819,6.295,148.197
C08054=1232.190,251.435,-61.033,-176.821,6.293,148.197
C08055=1232.195,251.186,-61.007,-176.824,6.291,148.197
C08056=1232.199,250.937,-60.981,-176.826,6.289,148.197
C08057=1232.204,250.689,-60.953,-176.829,6.287,148.198
C08058=1232.209,250.440,-60.927,-176.831,6.285,148.198
C08059=1232.212,250.192,-60.901,-176.834,6.284,148.198
C08060=1232.217,249.943,-60.874,-176.836,6.281,148.198
C08061=1232.222,249.695,-60.848,-176.839,6.279,148.199
C08062=1232.227,249.447,-60.821,-176.841,6.278,148.199
C08063=1232.231,249.198,-60.795,-176.844,6.276,148.199
C08064=1232.235,248.949,-60.768,-176.846,6.274,148.200
C08065=1232.240,248.700,-60.743,-176.849,6.272,148.200
C08066=1232.244,248.452,-60.716,-176.851,6.270,148.200
C08067=1232.249,248.203,-60.690,-176.854,6.268,148.200
C08068=1232.252,247.955,-60.663,-176.856,6.266,148.201
C08069=1232.257,247.706,-60.637,-176.859,6.264,148.201
C08070=1232.261,247.458,-60.610,-176.861,6.262,148.201
C08071=1232.266,247.209,-60.584,-176.864,6.260,148.201
C08072=1232.270,246.960,-60.558,-176.866,6.258,148.202
C08073=1232.276,246.712,-60.532,-176.869,6.256,148.202
C08074=1232.280,246.464,-60.505,-176.872,6.254,148.202
C08075=1232.284,246.215,-60.479,-176.874,6.253,148.203
C08076=1232.289,245.966,-60.453,-176.876,6.251,148.203
C08077=1232.293,245.718,-60.427,-176.878,6.249,148.203
C08078=1232.297,245.469,-60.401,-176.881,6.247,148.203
C08079=1232.302,245.220,-60.374,-176.884,6.245,148.204
C08080=1232.306,244.972,-60.348,-176.886,6.243,148.204
C08081=1232.311,244.723,-60.322,-176.889,6.242,148.204
C08082=1232.315,244.475,-60.296,-176.891,6.239,148.204
C08083=1232.320,244.226,-60.270,-176.893,6.237,148.205
C08084=1232.325,243.977,-60.244,-176.896,6.236,148.205
C08085=1232.329,243.729,-60.217,-176.899,6.234,148.205
C08086=1232.333,243.480,-60.191,-176.901,6.232,148.206
C08087=1232.338,243.232,-60.165,-176.904,6.230,148.206
C08088=1232.342,242.983,-60.139,-176.906,6.228,148.206
C08089=1232.346,242.735,-60.113,-176.909,6.226,148.206
C08090=1232.351,242.486,-60.087,-176.911,6.224,148.207
C08091=1232.356,242.237,-60.061,-176.914,6.222,148.207
C08092=1232.360,241.989,-60.035,-176.916,6.221,148.207
C08093=1232.364,241.740,-60.009,-176.919,6.219,148.208
C08094=1232.369,241.491,-59.983,-176.921,6.217,148.208
C08095=1232.374,241.243,-59.957,-176.923,6.215,148.208
C08096=1232.377,240.994,-59.931,-176.926,6.213,148.208
C08097=1232.382,240.746,-59.905,-176.929,6.211,148.209
C08098=1232.387,240.497,-59.879,-176.931,6.209,148.209
C08099=1232.392,240.248,-59.853,-176.934,6.208,148.209
C08100=1232.396,239.999,-59.827,-176.936,6.206,148.210
C08101=1232.401,239.751,-59.802,-176.939,6.204,148.210
C08102=1232.404,239.503,-59.776,-176.942,6.202,148.210
C08103=1232.409,239.254,-59.749,-176.944,6.200,148.210
C08104=1232.414,239.005,-59.723,-176.946,6.199,148.211
C08105=1232.418,238.756,-59.698,-176.948,6.197,148.211
C08106=1232.423,238.508,-59.672,-176.951,6.195,148.211
C08107=1232.427,238.260,-59.647,-176.954,6.193,148.212
C08108=1232.432,237.988,-59.619,-176.956,6.191,148.212
C08109=1232.437,237.717,-59.590,-176.959,6.188,148.212
C08110=1232.442,237.445,-59.562,-176.962,6.187,148.213
C08111=1232.447,237.174,-59.534,-176.965,6.185,148.213
C08112=1232.452,236.925,-59.508,-176.967,6.183,148.213
C08113=1232.456,236.676,-59.482,-176.970,6.181,148.214
C08114=1232.461,236.428,-59.457,-176.972,6.179,148.214
C08115=1232.465,236.179,-59.431,-176.975,6.177,148.214
C08116=1232.469,235.930,-59.405,-176.977,6.176,148.215
C08117=1232.474,235.682,-59.380,-176.980,6.174,148.215
C08118=1232.478,235.433,-59.354,-176.982,6.172,148.215
C08119=1232.483,235.184,-59.328,-176.985,6.170,148.215
C08120=1232.487,234.936,-59.302,-176.987,6.168,148.216
C08121=1232.492,234.687,-59.277,-176.990,6.166,148.216
C08122=1232.496,234.439,-59.251,-176.992,6.164,148.216
C08123=1232.501,234.190,-59.225,-176.995,6.163,148.217
C08124=1232.505,233.942,-59.200,-176.998,6.161,148.217
C08125=1232.510,233.693,-59.174,-177.000,6.160,148.217
C08126=1232.514,233.444,-59.148,-177.002,6.158,148.218
C08127=1232.519,233.195,-59.124,-177.005,6.156,148.218
C08128=1232.523,232.947,-59.098,-177.008,6.154,148.218
C08129=1232.528,232.698,-59.073,-177.010,6.152,148.218
C08130=1232.532,232.450,-59.047,-177.013,6.150,148.219
C08131=1232.536,232.201,-59.021,-177.015,6.148,148.219
C08132=1232.541,231.953,-58.996,-177.017,6.146,148.219
C08133=1232.546,231.703,-58.971,-177.020,6.145,148.220
C08134=1232.550,231.455,-58.945,-177.022,6.143,148.220
C08135=1232.555,231.206,-58.920,-177.025,6.141,148.220
C08136=1232.559,230.958,-58.894,-177.027,6.140,148.221
C08137=1232.564,230.710,-58.868,-177.030,6.138,148.221
C08138=1232.568,230.460,-58.843,-177.033,6.136,148.221
C08139=1232.573,230.211,-58.818,-177.035,6.134,148.221
C08140=1232.578,229.963,-58.792,-177.038,6.132,148.222
C08141=1232.582,229.714,-58.767,-177.040,6.131,148.222
C08142=1232.587,229.466,-58.742,-177.043,6.129,148.222
C08143=1232.590,229.217,-58.717,-177.045,6.127,148.223
C08144=1232.595,228.968,-58.691,-177.048,6.125,148.223
C08145=1232.600,228.720,-58.666,-177.050,6.123,148.223
C08146=1232.604,228.471,-58.641,-177.053,6.122,148.224
C08147=1232.609,228.223,-58.615,-177.056,6.120,148.224
C08148=1232.613,227.973,-58.590,-177.058,6.119,148.224
C08149=1232.618,227.725,-58.565,-177.060,6.117,148.225
C08150=1232.623,227.476,-58.540,-177.063,6.115,148.225
C08151=1232.627,227.228,-58.515,-177.066,6.113,148.225
C08152=1232.631,226.979,-58.489,-177.068,6.111,148.226
C08153=1232.636,226.730,-58.464,-177.071,6.109,148.226
C08154=1232.640,226.482,-58.439,-177.073,6.107,148.226
C08155=1232.645,226.232,-58.414,-177.076,6.106,148.227
C08156=1232.650,225.984,-58.388,-177.078,6.105,148.227
C08157=1232.653,225.735,-58.364,-177.081,6.103,148.227
C08158=1232.658,225.487,-58.338,-177.083,6.101,148.228
C08159=1232.663,225.237,-58.313,-177.086,6.099,148.228
C08160=1232.668,224.989,-58.288,-177.088,6.097,148.228
C08161=1232.672,224.740,-58.263,-177.091,6.095,148.228
C08162=1232.676,224.492,-58.238,-177.093,6.094,148.229
C08163=1232.681,224.243,-58.213,-177.095,6.092,148.229
C08164=1232.686,223.995,-58.188,-177.098,6.090,148.229
C08165=1232.690,223.745,-58.163,-177.101,6.088,148.230
C08166=1232.695,223.497,-58.137,-177.103,6.086,148.230
C08167=1232.699,223.248,-58.113,-177.106,6.084,148.230
C08168=1232.704,223.000,-58.088,-177.108,6.083,148.231
C08169=1232.708,222.750,-58.063,-177.111,6.082,148.231
C08170=1232.712,222.503,-58.038,-177.114,6.080,148.232
C08171=1232.717,222.254,-58.013,-177.116,6.078,148.232
C08172=1232.722,222.005,-57.988,-177.119,6.076,148.232
C08173=1232.727,221.756,-57.963,-177.122,6.074,148.233
C08174=1232.731,221.507,-57.938,-177.124,6.073,148.233
C08175=1232.736,221.259,-57.914,-177.126,6.071,148.233
C08176=1232.740,221.010,-57.888,-177.129,6.070,148.234
C08177=1232.744,220.761,-57.864,-177.132,6.068,148.234
C08178=1232.749,220.512,-57.839,-177.134,6.066,148.234
C08179=1232.754,220.264,-57.813,-177.137,6.064,148.235
C08180=1232.758,220.015,-57.789,-177.139,6.063,148.235
C08181=1232.763,219.766,-57.764,-177.141,6.061,148.235
C08182=1232.767,219.518,-57.739,-177.144,6.059,148.236
C08183=1232.771,219.269,-57.714,-177.147,6.057,148.236
C08184=1232.776,219.020,-57.690,-177.149,6.055,148.236
C08185=1232.781,218.772,-57.666,-177.152,6.054,148.237
C08186=1232.785,218.523,-57.640,-177.154,6.053,148.237
C08187=1232.790,218.274,-57.615,-177.157,6.051,148.237
C08188=1232.794,218.025,-57.591,-177.159,6.049,148.238
C08189=1232.799,217.776,-57.566,-177.162,6.047,148.238
C08190=1232.803,217.528,-57.542,-177.165,6.045,148.238
C08191=1232.808,217.279,-57.516,-177.167,6.044,148.239
C08192=1232.812,217.031,-57.492,-177.169,6.042,148.239
C08193=1232.817,216.782,-57.468,-177.172,6.040,148.239
C08194=1232.822,216.533,-57.442,-177.175,6.038,148.240
C08195=1232.826,216.284,-57.418,-177.178,6.037,148.240
C08196=1232.831,216.035,-57.393,-177.180,6.035,148.241
C08197=1232.835,215.787,-57.369,-177.182,6.034,148.241
C08198=1232.840,215.538,-57.344,-177.185,6.032,148.241
C08199=1232.844,215.289,-57.319,-177.188,6.030,148.242
C08200=1232.849,215.040,-57.295,-177.190,6.028,148.242
C08201=1232.853,214.792,-57.271,-177.193,6.027,148.242
C08202=1232.858,214.542,-57.246,-177.195,6.025,148.243
C08203=1232.862,214.294,-57.222,-177.198,6.024,148.243
C08204=1232.867,214.045,-57.197,-177.200,6.022,148.243
C08205=1232.871,213.796,-57.173,-177.203,6.020,148.244
C08206=1232.876,213.548,-57.148,-177.205,6.018,148.244
C08207=1232.880,213.299,-57.124,-177.207,6.017,148.244
C08208=1232.886,213.050,-57.099,-177.210,6.015,148.245
C08209=1232.889,212.801,-57.075,-177.213,6.014,148.245
C08210=1232.894,212.553,-57.051,-177.216,6.012,148.246
C08211=1232.899,212.304,-57.026,-177.218,6.010,148.246
C08212=1232.903,212.033,-56.999,-177.221,6.008,148.246
C08213=1232.909,211.763,-56.972,-177.224,6.006,148.247
C08214=1232.913,211.493,-56.947,-177.227,6.005,148.247
C08215=1232.919,211.222,-56.920,-177.229,6.003,148.247
C08216=1232.924,210.974,-56.895,-177.232,6.002,148.248
C08217=1232.927,210.725,-56.871,-177.234,6.000,148.248
C08218=1232.932,210.476,-56.847,-177.237,5.998,148.248
C08219=1232.937,210.227,-56.822,-177.239,5.996,148.249
C08220=1232.941,209.979,-56.798,-177.242,5.995,148.249
C08221=1232.945,209.729,-56.774,-177.244,5.993,148.249
C08222=1232.951,209.481,-56.750,-177.247,5.992,148.250
C08223=1232.955,209.232,-56.726,-177.250,5.990,148.250
C08224=1232.959,208.984,-56.702,-177.253,5.988,148.251
C08225=1232.964,208.734,-56.676,-177.255,5.987,148.251
C08226=1232.968,208.486,-56.652,-177.257,5.985,148.251
C08227=1232.973,208.237,-56.629,-177.260,5.983,148.252
C08228=1232.978,207.988,-56.604,-177.262,5.981,148.252
C08229=1232.983,207.740,-56.580,-177.265,5.980,148.252
C08230=1232.986,207.491,-56.556,-177.267,5.978,148.253
C08231=1232.992,207.241,-56.532,-177.270,5.977,148.253
C08232=1232.996,206.993,-56.508,-177.273,5.975,148.254
C08233=1233.001,206.744,-56.484,-177.275,5.974,148.254
C08234=1233.006,206.496,-56.459,-177.278,5.972,148.254
C08235=1233.010,206.246,-56.435,-177.280,5.970,148.255
C08236=1233.014,205.998,-56.411,-177.283,5.968,148.255
C08237=1233.019,205.749,-56.387,-177.285,5.967,148.255
C08238=1233.024,205.500,-56.363,-177.288,5.965,148.256
C08239=1233.028,205.251,-56.339,-177.291,5.964,148.256
C08240=1233.033,205.003,-56.315,-177.293,5.962,148.257
C08241=1233.037,204.753,-56.291,-177.295,5.961,148.257
C08242=1233.041,204.505,-56.267,-177.298,5.959,148.257
C08243=1233.046,204.256,-56.243,-177.301,5.957,148.258
C08244=1233.051,204.007,-56.219,-177.303,5.955,148.258
C08245=1233.056,203.759,-56.195,-177.305,5.954,148.258
C08246=1233.060,203.510,-56.171,-177.309,5.953,148.259
C08247=1233.065,203.261,-56.148,-177.311,5.951,148.259
C08248=1233.069,203.012,-56.123,-177.313,5.950,148.260
C08249=1233.074,202.763,-56.099,-177.316,5.948,148.260
C08250=1233.078,202.514,-56.075,-177.319,5.946,148.260
C08251=1233.083,202.265,-56.052,-177.321,5.944,148.261
C08252=1233.087,202.017,-56.028,-177.323,5.943,148.261
C08253=1233.092,201.769,-56.004,-177.326,5.942,148.262
C08254=1233.096,201.520,-55.980,-177.329,5.940,148.262
C08255=1233.102,201.271,-55.956,-177.331,5.939,148.262
C08256=1233.106,201.022,-55.932,-177.334,5.937,148.263
C08257=1233.111,200.773,-55.908,-177.336,5.935,148.263
C08258=1233.115,200.524,-55.885,-177.339,5.933,148.263
C08259=1233.119,200.275,-55.861,-177.341,5.932,148.264
C08260=1233.124,200.026,-55.837,-177.344,5.931,148.264
C08261=1233.129,199.777,-55.814,-177.347,5.929,148.265
C08262=1233.133,199.529,-55.790,-177.349,5.928,148.265
C08263=1233.138,199.280,-55.766,-177.352,5.926,148.265
C08264=1233.142,199.031,-55.742,-177.354,5.924,148.266
C08265=1233.147,198.782,-55.719,-177.357,5.922,148.266
C08266=1233.151,198.533,-55.696,-177.359,5.922,148.267
C08267=1233.156,198.285,-55.672,-177.362,5.920,148.267
C08268=1233.161,198.036,-55.648,-177.365,5.918,148.267
C08269=1233.166,197.787,-55.624,-177.367,5.917,148.268
C08270=1233.170,197.538,-55.600,-177.369,5.915,148.268
C08271=1233.175,197.289,-55.577,-177.372,5.914,148.269
C08272=1233.179,197.041,-55.553,-177.375,5.913,148.269
C08273=1233.184,196.792,-55.529,-177.377,5.911,148.269
C08274=1233.189,196.543,-55.506,-177.380,5.909,148.270
C08275=1233.193,196.294,-55.482,-177.382,5.908,148.270
C08276=1233.198,196.045,-55.459,-177.385,5.906,148.270
C08277=1233.202,195.796,-55.436,-177.388,5.904,148.271
C08278=1233.207,195.547,-55.412,-177.390,5.903,148.271
C08279=1233.211,195.299,-55.388,-177.392,5.902,148.272
C08280=1233.216,195.050,-55.365,-177.395,5.900,148.272
C08281=1233.220,194.801,-55.342,-177.397,5.899,148.272
C08282=1233.225,194.552,-55.318,-177.400,5.897,148.273
C08283=1233.229,194.303,-55.294,-177.403,5.895,148.273
C08284=1233.234,194.054,-55.271,-177.405,5.894,148.274
C08285=1233.239,193.805,-55.248,-177.408,5.892,148.274
C08286=1233.244,193.556,-55.224,-177.410,5.891,148.274
C08287=1233.248,193.307,-55.201,-177.413,5.890,148.275
C08288=1233.253,193.059,-55.177,-177.415,5.888,148.275
C08289=1233.257,192.810,-55.153,-177.418,5.886,148.276
C08290=1233.262,192.561,-55.130,-177.420,5.885,148.276
C08291=1233.266,192.312,-55.107,-177.423,5.883,148.276
C08292=1233.271,192.063,-55.084,-177.426,5.882,148.277
C08293=1233.275,191.814,-55.061,-177.428,5.881,148.277
C08294=1233.280,191.565,-55.037,-177.431,5.879,148.278
C08295=1233.285,191.317,-55.014,-177.433,5.877,148.278
C08296=1233.290,191.068,-54.990,-177.435,5.876,148.278
C08297=1233.295,190.819,-54.967,-177.439,5.875,148.279
C08298=1233.298,190.570,-54.944,-177.441,5.873,148.279
C08299=1233.303,190.321,-54.921,-177.443,5.872,148.280
C08300=1233.308,190.072,-54.897,-177.446,5.870,148.280
C08301=1233.313,189.823,-54.874,-177.449,5.868,148.281
C08302=1233.317,189.574,-54.851,-177.451,5.867,148.281
C08303=1233.321,189.326,-54.828,-177.454,5.865,148.281
C08304=1233.326,189.077,-54.804,-177.456,5.864,148.282
C08305=1233.331,188.828,-54.781,-177.458,5.863,148.282
C08306=1233.336,188.579,-54.758,-177.462,5.861,148.283
C08307=1233.340,188.330,-54.735,-177.464,5.860,148.283
C08308=1233.345,188.081,-54.712,-177.466,5.858,148.283
C08309=1233.349,187.832,-54.689,-177.469,5.856,148.284
C08310=1233.354,187.583,-54.665,-177.472,5.856,148.284
C08311=1233.358,187.335,-54.642,-177.474,5.854,148.285
C08312=1233.363,187.086,-54.619,-177.476,5.853,148.285
C08313=1233.368,186.837,-54.596,-177.479,5.851,148.285
C08314=1233.373,186.588,-54.573,-177.482,5.849,148.286
C08315=1233.377,186.339,-54.551,-177.484,5.848,148.286
C08316=1233.382,186.069,-54.526,-177.487,5.846,148.287
C08317=1233.387,185.800,-54.500,-177.490,5.845,148.287
C08318=1233.392,185.531,-54.475,-177.493,5.843,148.288
C08319=1233.397,185.261,-54.450,-177.496,5.842,148.288
C08320=1233.402,185.012,-54.427,-177.498,5.841,148.289
C08321=1233.406,184.762,-54.405,-177.500,5.839,148.289
C08322=1233.411,184.513,-54.382,-177.503,5.838,148.289
C08323=1233.416,184.264,-54.358,-177.506,5.836,148.290
C08324=1233.420,184.016,-54.336,-177.508,5.834,148.290
C08325=1233.425,183.767,-54.313,-177.510,5.833,148.291
C08326=1233.430,183.518,-54.290,-177.513,5.831,148.291
C08327=1233.434,183.269,-54.267,-177.516,5.831,148.292
C08328=1233.439,183.021,-54.244,-177.518,5.829,148.292
C08329=1233.443,182.772,-54.221,-177.521,5.827,148.292
C08330=1233.448,182.522,-54.199,-177.523,5.826,148.293
C08331=1233.453,182.273,-54.175,-177.526,5.825,148.293
C08332=1233.457,182.024,-54.153,-177.528,5.824,148.294
C08333=1233.462,181.776,-54.130,-177.531,5.822,148.294
C08334=1233.466,181.527,-54.108,-177.534,5.820,148.295
C08335=1233.471,181.278,-54.084,-177.536,5.819,148.295
C08336=1233.476,181.029,-54.061,-177.539,5.817,148.295
C08337=1233.481,180.780,-54.039,-177.541,5.816,148.296
C08338=1233.485,180.531,-54.016,-177.544,5.815,148.296
C08339=1233.489,180.282,-53.993,-177.547,5.813,148.297
C08340=1233.494,180.033,-53.970,-177.549,5.812,148.297
C08341=1233.499,179.785,-53.948,-177.552,5.810,148.298
C08342=1233.503,179.536,-53.925,-177.554,5.809,148.298
C08343=1233.508,179.286,-53.903,-177.557,5.808,148.298
C08344=1233.513,179.038,-53.880,-177.559,5.807,148.299
C08345=1233.517,178.789,-53.858,-177.562,5.805,148.299
C08346=1233.522,178.540,-53.834,-177.564,5.803,148.300
C08347=1233.526,178.291,-53.811,-177.567,5.802,148.300
C08348=1233.532,178.042,-53.789,-177.570,5.801,148.301
C08349=1233.536,177.793,-53.766,-177.572,5.800,148.301
C08350=1233.541,177.544,-53.744,-177.574,5.798,148.301
C08351=1233.545,177.296,-53.721,-177.576,5.797,148.302
C08352=1233.550,177.046,-53.699,-177.580,5.795,148.302
C08353=1233.554,176.797,-53.676,-177.582,5.794,148.303
C08354=1233.560,176.548,-53.654,-177.584,5.792,148.303
C08355=1233.564,176.299,-53.631,-177.587,5.791,148.304
C08356=1233.568,176.050,-53.609,-177.590,5.790,148.304
C08357=1233.573,175.802,-53.586,-177.592,5.788,148.304
C08358=1233.577,175.552,-53.564,-177.595,5.787,148.305
C08359=1233.582,175.303,-53.540,-177.597,5.786,148.305
C08360=1233.587,175.055,-53.519,-177.600,5.785,148.306
C08361=1233.592,174.805,-53.496,-177.602,5.783,148.306
C08362=1233.596,174.556,-53.473,-177.605,5.782,148.307
C08363=1233.601,174.308,-53.452,-177.607,5.780,148.307
C08364=1233.606,174.059,-53.428,-177.610,5.779,148.307
C08365=1233.610,173.810,-53.407,-177.613,5.778,148.308
C08366=1233.614,173.561,-53.384,-177.615,5.776,148.308
C08367=1233.619,173.312,-53.361,-177.617,5.775,148.309
C08368=1233.624,173.063,-53.340,-177.621,5.773,148.309
C08369=1233.628,172.814,-53.317,-177.623,5.772,148.310
C08370=1233.633,172.565,-53.294,-177.625,5.770,148.310
C08371=1233.638,172.316,-53.272,-177.628,5.770,148.311
C08372=1233.642,172.067,-53.250,-177.631,5.768,148.311
C08373=1233.648,171.818,-53.227,-177.633,5.767,148.311
C08374=1233.652,171.569,-53.205,-177.636,5.765,148.312
C08375=1233.657,171.321,-53.183,-177.638,5.764,148.312
C08376=1233.662,171.071,-53.160,-177.640,5.763,148.313
C08377=1233.666,170.822,-53.138,-177.643,5.762,148.313
C08378=1233.671,170.573,-53.117,-177.646,5.760,148.314
C08379=1233.675,170.324,-53.093,-177.648,5.759,148.314
C08380=1233.680,170.076,-53.072,-177.651,5.758,148.315
C08381=1233.685,169.826,-53.050,-177.653,5.757,148.315
C08382=1233.689,169.578,-53.028,-177.656,5.755,148.315
C08383=1233.694,169.329,-53.004,-177.658,5.754,148.316
C08384=1233.699,169.080,-52.983,-177.661,5.752,148.316
C08385=1233.703,168.831,-52.961,-177.663,5.751,148.317
C08386=1233.707,168.581,-52.939,-177.666,5.750,148.317
C08387=1233.713,168.332,-52.916,-177.668,5.749,148.318
C08388=1233.717,168.083,-52.894,-177.671,5.747,148.318
C08389=1233.722,167.835,-52.872,-177.674,5.746,148.319
C08390=1233.726,167.586,-52.850,-177.676,5.744,148.319
C08391=1233.731,167.337,-52.828,-177.679,5.744,148.320
C08392=1233.736,167.087,-52.806,-177.681,5.742,148.320
C08393=1233.741,166.839,-52.784,-177.683,5.741,148.320
C08394=1233.745,166.589,-52.762,-177.687,5.739,148.321
C08395=1233.750,166.341,-52.740,-177.689,5.738,148.321
C08396=1233.754,166.092,-52.718,-177.691,5.736,148.322
C08397=1233.759,165.843,-52.696,-177.694,5.736,148.322
C08398=1233.764,165.594,-52.673,-177.697,5.734,148.323
C08399=1233.769,165.345,-52.651,-177.699,5.733,148.323
C08400=1233.773,165.096,-52.629,-177.702,5.731,148.324
C08401=1233.778,164.847,-52.608,-177.704,5.730,148.324
C08402=1233.782,164.598,-52.586,-177.707,5.729,148.325
C08403=1233.787,164.349,-52.564,-177.709,5.728,148.325
C08404=1233.791,164.100,-52.542,-177.712,5.726,148.326
C08405=1233.796,163.851,-52.520,-177.714,5.725,148.326
C08406=1233.801,163.602,-52.498,-177.717,5.724,148.327
C08407=1233.806,163.353,-52.476,-177.719,5.723,148.327
C08408=1233.811,163.104,-52.454,-177.722,5.721,148.327
C08409=1233.815,162.855,-52.432,-177.724,5.720,148.328
C08410=1233.820,162.606,-52.410,-177.728,5.719,148.328
C08411=1233.824,162.357,-52.388,-177.730,5.718,148.329
C08412=1233.829,162.108,-52.367,-177.732,5.716,148.329
C08413=1233.834,161.858,-52.345,-177.735,5.715,148.330
C08414=1233.839,161.610,-52.324,-177.737,5.714,148.330
C08415=1233.844,161.361,-52.302,-177.740,5.713,148.331
C08416=1233.848,161.112,-52.280,-177.742,5.712,148.331
C08417=1233.853,160.863,-52.258,-177.745,5.710,148.332
C08418=1233.857,160.614,-52.236,-177.748,5.709,148.332
C08419=1233.862,160.365,-52.215,-177.750,5.707,148.333
C08420=1233.867,160.096,-52.191,-177.753,5.707,148.333
C08421=1233.872,159.827,-52.167,-177.755,5.705,148.334
C08422=1233.877,159.558,-52.144,-177.759,5.703,148.334
C08423=1233.883,159.289,-52.121,-177.761,5.703,148.335
C08424=1233.887,159.039,-52.099,-177.764,5.701,148.335
C08425=1233.892,158.791,-52.077,-177.766,5.700,148.336
C08426=1233.896,158.541,-52.055,-177.769,5.698,148.336
C08427=1233.901,158.292,-52.034,-177.771,5.697,148.337
C08428=1233.906,158.043,-52.013,-177.774,5.696,148.337
C08429=1233.910,157.794,-51.991,-177.776,5.695,148.337
C08430=1233.915,157.545,-51.969,-177.779,5.694,148.338
C08431=1233.920,157.297,-51.947,-177.782,5.692,148.338
C08432=1233.924,157.047,-51.926,-177.784,5.691,148.339
C08433=1233.929,156.799,-51.905,-177.787,5.690,148.339
C08434=1233.934,156.550,-51.883,-177.789,5.689,148.340
C08435=1233.938,156.300,-51.862,-177.792,5.687,148.340
C08436=1233.943,156.051,-51.840,-177.794,5.686,148.341
C08437=1233.948,155.803,-51.818,-177.796,5.685,148.341
C08438=1233.953,155.553,-51.797,-177.800,5.684,148.342
C08439=1233.957,155.304,-51.775,-177.802,5.683,148.342
C08440=1233.962,155.055,-51.754,-177.805,5.681,148.343
C08441=1233.967,154.805,-51.732,-177.807,5.680,148.343
C08442=1233.971,154.557,-51.711,-177.810,5.678,148.344
C08443=1233.976,154.308,-51.690,-177.812,5.678,148.344
C08444=1233.980,154.058,-51.668,-177.814,5.677,148.345
C08445=1233.985,153.810,-51.647,-177.817,5.675,148.345
C08446=1233.990,153.561,-51.625,-177.819,5.674,148.346
C08447=1233.995,153.312,-51.604,-177.823,5.673,148.346
C08448=1233.999,153.063,-51.582,-177.825,5.672,148.347
C08449=1234.004,152.814,-51.562,-177.827,5.671,148.347
C08450=1234.009,152.565,-51.540,-177.830,5.669,148.348
C08451=1234.014,152.316,-51.519,-177.832,5.668,148.348
C08452=1234.018,152.066,-51.497,-177.835,5.667,148.349
C08453=1234.023,151.817,-51.476,-177.837,5.666,148.349
C08454=1234.028,151.569,-51.455,-177.840,5.665,148.350
C08455=1234.033,151.320,-51.433,-177.843,5.663,148.350
C08456=1234.037,151.070,-51.412,-177.845,5.663,148.351
C08457=1234.042,150.822,-51.390,-177.848,5.661,148.351
C08458=1234.046,150.573,-51.370,-177.850,5.660,148.352
C08459=1234.052,150.323,-51.349,-177.853,5.659,148.352
C08460=1234.056,150.074,-51.327,-177.856,5.658,148.353
C08461=1234.061,149.825,-51.306,-177.858,5.657,148.353
C08462=1234.065,149.576,-51.285,-177.860,5.655,148.353
C08463=1234.070,149.327,-51.264,-177.863,5.654,148.354
C08464=1234.075,149.078,-51.242,-177.865,5.653,148.354
C08465=1234.079,148.829,-51.221,-177.868,5.652,148.355
C08466=1234.084,148.580,-51.200,-177.870,5.651,148.355
C08467=1234.089,148.331,-51.179,-177.874,5.649,148.356
C08468=1234.094,148.082,-51.158,-177.876,5.648,148.356
C08469=1234.098,147.833,-51.136,-177.878,5.648,148.357
C08470=1234.103,147.583,-51.115,-177.881,5.646,148.357
C08471=1234.108,147.334,-51.094,-177.884,5.645,148.358
C08472=1234.112,147.086,-51.073,-177.886,5.644,148.358
C08473=1234.118,146.837,-51.052,-177.889,5.643,148.359
C08474=1234.122,146.587,-51.030,-177.891,5.642,148.359
C08475=1234.126,146.338,-51.010,-177.894,5.640,148.360
C08476=1234.131,146.089,-50.989,-177.896,5.639,148.360
C08477=1234.136,145.840,-50.968,-177.898,5.638,148.361
C08478=1234.141,145.591,-50.947,-177.901,5.637,148.361
C08479=1234.146,145.342,-50.926,-177.903,5.636,148.362
C08480=1234.150,145.093,-50.905,-177.906,5.635,148.362
C08481=1234.155,144.844,-50.883,-177.909,5.633,148.363
C08482=1234.160,144.595,-50.862,-177.911,5.633,148.363
C08483=1234.164,144.346,-50.842,-177.913,5.632,148.364
C08484=1234.169,144.096,-50.821,-177.917,5.630,148.364
C08485=1234.173,143.848,-50.800,-177.919,5.629,148.365
C08486=1234.179,143.599,-50.779,-177.922,5.628,148.365
C08487=1234.183,143.350,-50.759,-177.924,5.627,148.366
C08488=1234.188,143.100,-50.737,-177.927,5.626,148.366
C08489=1234.193,142.851,-50.716,-177.929,5.624,148.367
C08490=1234.197,142.602,-50.695,-177.932,5.623,148.367
C08491=1234.202,142.353,-50.674,-177.934,5.622,148.368
C08492=1234.207,142.104,-50.654,-177.937,5.621,148.368
C08493=1234.212,141.855,-50.633,-177.939,5.620,148.369
C08494=1234.216,141.606,-50.613,-177.942,5.619,148.370
C08495=1234.221,141.357,-50.592,-177.944,5.618,148.370
C08496=1234.226,141.108,-50.570,-177.947,5.617,148.371
C08497=1234.231,140.859,-50.550,-177.949,5.616,148.371
C08498=1234.235,140.609,-50.529,-177.952,5.614,148.372
C08499=1234.240,140.360,-50.508,-177.954,5.613,148.372
C08500=1234.244,140.111,-50.487,-177.957,5.613,148.373
C08501=1234.249,139.862,-50.466,-177.960,5.611,148.373
C08502=1234.254,139.613,-50.446,-177.962,5.610,148.374
C08503=1234.259,139.364,-50.425,-177.964,5.609,148.374
C08504=1234.263,139.115,-50.405,-177.968,5.608,148.375
C08505=1234.269,138.866,-50.384,-177.970,5.607,148.375
C08506=1234.273,138.617,-50.363,-177.972,5.606,148.376
C08507=1234.277,138.368,-50.343,-177.975,5.605,148.376
C08508=1234.283,138.118,-50.322,-177.978,5.604,148.377
C08509=1234.287,137.869,-50.302,-177.980,5.603,148.377
C08510=1234.292,137.620,-50.281,-177.983,5.601,148.378
C08511=1234.297,137.371,-50.260,-177.985,5.601,148.378
C08512=1234.302,137.122,-50.239,-177.988,5.600,148.379
C08513=1234.306,136.873,-50.219,-177.991,5.598,148.379
C08514=1234.311,136.624,-50.199,-177.993,5.597,148.380
C08515=1234.316,136.375,-50.178,-177.995,5.596,148.380
C08516=1234.320,136.126,-50.157,-177.998,5.596,148.381
C08517=1234.325,135.877,-50.137,-178.001,5.594,148.381
C08518=1234.330,135.628,-50.116,-178.003,5.593,148.382
C08519=1234.334,135.379,-50.096,-178.005,5.592,148.382
C08520=1234.340,135.129,-50.075,-178.008,5.591,148.383
C08521=1234.344,134.881,-50.054,-178.011,5.590,148.383
C08522=1234.348,134.632,-50.034,-178.013,5.589,148.384
C08523=1234.354,134.382,-50.014,-178.016,5.587,148.384
C08524=1234.358,134.114,-49.992,-178.019,5.587,148.385
C08525=1234.363,133.845,-49.969,-178.022,5.585,148.386
C08526=1234.369,133.576,-49.947,-178.024,5.584,148.386
C08527=1234.374,133.307,-49.925,-178.027,5.583,148.387
C08528=1234.379,133.058,-49.905,-178.030,5.582,148.387
C08529=1234.383,132.809,-49.885,-178.032,5.581,148.388
C08530=1234.388,132.560,-49.865,-178.034,5.581,148.388
C08531=1234.393,132.311,-49.844,-178.037,5.579,148.389
C08532=1234.397,132.062,-49.823,-178.040,5.578,148.389
C08533=1234.402,131.813,-49.803,-178.042,5.577,148.390
C08534=1234.407,131.563,-49.783,-178.045,5.576,148.390
C08535=1234.412,131.314,-49.762,-178.047,5.575,148.391
C08536=1234.416,131.065,-49.742,-178.050,5.574,148.391
C08537=1234.421,130.816,-49.722,-178.052,5.573,148.392
C08538=1234.427,130.567,-49.702,-178.055,5.572,148.392
C08539=1234.431,130.318,-49.681,-178.057,5.571,148.393
C08540=1234.436,130.069,-49.661,-178.060,5.570,148.393
C08541=1234.440,129.820,-49.641,-178.063,5.568,148.394
C08542=1234.446,129.570,-49.620,-178.065,5.568,148.395
C08543=1234.450,129.321,-49.600,-178.067,5.567,148.395
C08544=1234.454,129.072,-49.580,-178.070,5.566,148.396
C08545=1234.459,128.823,-49.560,-178.073,5.564,148.396
C08546=1234.464,128.574,-49.540,-178.075,5.564,148.397
C08547=1234.468,128.325,-49.519,-178.077,5.563,148.397
C08548=1234.474,128.076,-49.499,-178.080,5.562,148.398
C08549=1234.479,127.827,-49.479,-178.083,5.561,148.398
C08550=1234.483,127.577,-49.459,-178.085,5.560,148.399
C08551=1234.488,127.328,-49.439,-178.088,5.559,148.399
C08552=1234.492,127.079,-49.418,-178.090,5.558,148.400
C08553=1234.497,126.830,-49.399,-178.093,5.557,148.400
C08554=1234.502,126.580,-49.378,-178.095,5.556,148.401
C08555=1234.507,126.331,-49.359,-178.098,5.555,148.401
C08556=1234.512,126.082,-49.338,-178.101,5.554,148.402
C08557=1234.516,125.834,-49.318,-178.103,5.553,148.402
C08558=1234.521,125.584,-49.298,-178.106,5.552,148.403
C08559=1234.526,125.335,-49.278,-178.108,5.551,148.404
C08560=1234.530,125.085,-49.258,-178.111,5.550,148.404
C08561=1234.535,124.837,-49.238,-178.114,5.549,148.405
C08562=1234.540,124.588,-49.218,-178.116,5.548,148.405
C08563=1234.545,124.338,-49.198,-178.118,5.547,148.406
C08564=1234.550,124.089,-49.178,-178.121,5.546,148.406
C08565=1234.554,123.840,-49.157,-178.124,5.545,148.407
C08566=1234.559,123.590,-49.138,-178.126,5.544,148.408
C08567=1234.564,123.342,-49.118,-178.128,5.543,148.408
C08568=1234.569,123.092,-49.098,-178.131,5.542,148.409
C08569=1234.573,122.843,-49.078,-178.134,5.541,148.409
C08570=1234.578,122.594,-49.058,-178.136,5.540,148.410
C08571=1234.583,122.344,-49.038,-178.139,5.539,148.410
C08572=1234.588,122.096,-49.018,-178.141,5.538,148.411
C08573=1234.593,121.847,-48.999,-178.144,5.537,148.411
C08574=1234.597,121.598,-48.978,-178.146,5.536,148.412
C08575=1234.602,121.348,-48.959,-178.149,5.535,148.412
C08576=1234.607,121.099,-48.940,-178.152,5.535,148.413
C08577=1234.612,120.850,-48.919,-178.154,5.534,148.413
C08578=1234.616,120.601,-48.899,-178.157,5.532,148.414
C08579=1234.621,120.352,-48.879,-178.159,5.532,148.415
C08580=1234.626,120.103,-48.860,-178.162,5.531,148.415
C08581=1234.631,119.853,-48.840,-178.164,5.530,148.416
C08582=1234.635,119.604,-48.820,-178.167,5.528,148.416
C08583=1234.640,119.355,-48.800,-178.169,5.528,148.417
C08584=1234.645,119.106,-48.781,-178.172,5.527,148.417
C08585=1234.650,118.856,-48.761,-178.174,5.526,148.418
C08586=1234.655,118.607,-48.741,-178.177,5.525,148.418
C08587=1234.660,118.358,-48.722,-178.180,5.524,148.419
C08588=1234.665,118.109,-48.702,-178.182,5.523,148.419
C08589=1234.669,117.860,-48.681,-178.185,5.522,148.420
C08590=1234.673,117.611,-48.662,-178.187,5.521,148.420
C08591=1234.678,117.362,-48.643,-178.189,5.521,148.421
C08592=1234.683,117.112,-48.623,-178.193,5.519,148.422
C08593=1234.688,116.863,-48.603,-178.195,5.518,148.422
C08594=1234.693,116.614,-48.584,-178.197,5.518,148.423
C08595=1234.698,116.365,-48.564,-178.200,5.517,148.423
C08596=1234.702,116.115,-48.545,-178.202,5.516,148.424
C08597=1234.708,115.866,-48.525,-178.205,5.514,148.424
C08598=1234.712,115.618,-48.505,-178.208,5.514,148.425
C08599=1234.716,115.368,-48.486,-178.210,5.513,148.425
C08600=1234.722,115.119,-48.467,-178.213,5.512,148.426
C08601=1234.726,114.870,-48.447,-178.215,5.512,148.427
C08602=1234.731,114.620,-48.427,-178.218,5.510,148.427
C08603=1234.736,114.371,-48.408,-178.220,5.509,148.428
C08604=1234.741,114.122,-48.388,-178.223,5.508,148.428
C08605=1234.746,113.873,-48.368,-178.225,5.508,148.429
C08606=1234.750,113.624,-48.349,-178.228,5.507,148.430
C08607=1234.755,113.375,-48.330,-178.230,5.505,148.430
C08608=1234.760,113.125,-48.310,-178.233,5.505,148.431
C08609=1234.765,112.876,-48.291,-178.236,5.504,148.431
C08610=1234.770,112.627,-48.271,-178.238,5.503,148.432
C08611=1234.774,112.377,-48.252,-178.240,5.502,148.432
C08612=1234.779,112.129,-48.233,-178.243,5.502,148.433
C08613=1234.784,111.879,-48.213,-178.246,5.500,148.433
C08614=1234.789,111.630,-48.194,-178.248,5.499,148.434
C08615=1234.793,111.381,-48.175,-178.251,5.499,148.435
C08616=1234.798,111.131,-48.155,-178.253,5.498,148.435
C08617=1234.803,110.882,-48.136,-178.256,5.497,148.436
C08618=1234.808,110.633,-48.116,-178.258,5.496,148.436
C08619=1234.813,110.384,-48.097,-178.261,5.495,148.437
C08620=1234.817,110.135,-48.078,-178.264,5.494,148.437
C08621=1234.822,109.885,-48.058,-178.266,5.493,148.438
C08622=1234.827,109.636,-48.039,-178.268,5.492,148.438
C08623=1234.831,109.387,-48.020,-178.271,5.492,148.439
C08624=1234.837,109.138,-48.000,-178.273,5.491,148.440
C08625=1234.842,108.889,-47.981,-178.276,5.489,148.440
C08626=1234.846,108.640,-47.962,-178.279,5.489,148.441
C08627=1234.851,108.391,-47.942,-178.281,5.488,148.441
C08628=1234.856,108.122,-47.921,-178.284,5.487,148.442
C08629=1234.861,107.854,-47.900,-178.287,5.486,148.443
C08630=1234.867,107.585,-47.880,-178.289,5.485,148.443
C08631=1234.872,107.317,-47.859,-178.292,5.484,148.444
C08632=1234.876,107.067,-47.840,-178.295,5.484,148.444
C08633=1234.881,106.819,-47.821,-178.297,5.483,148.445
C08634=1234.886,106.569,-47.801,-178.300,5.481,148.445
C08635=1234.890,106.320,-47.782,-178.302,5.481,148.446
C08636=1234.896,106.070,-47.764,-178.305,5.480,148.447
C08637=1234.901,105.821,-47.744,-178.307,5.479,148.447
C08638=1234.905,105.572,-47.725,-178.310,5.478,148.448
C08639=1234.910,105.323,-47.706,-178.312,5.478,148.448
C08640=1234.915,105.074,-47.687,-178.315,5.477,148.449
C08641=1234.920,104.824,-47.668,-178.318,5.475,148.449
C08642=1234.925,104.575,-47.649,-178.320,5.475,148.450
C08643=1234.929,104.326,-47.630,-178.323,5.474,148.451
C08644=1234.934,104.077,-47.610,-178.325,5.473,148.451
C08645=1234.938,103.828,-47.591,-178.328,5.473,148.452
C08646=1234.944,103.578,-47.573,-178.330,5.472,148.452
C08647=1234.948,103.329,-47.554,-178.332,5.471,148.453
C08648=1234.953,103.080,-47.534,-178.336,5.470,148.453
C08649=1234.958,102.830,-47.516,-178.338,5.469,148.454
C08650=1234.963,102.581,-47.497,-178.341,5.468,148.455
C08651=1234.968,102.332,-47.478,-178.343,5.467,148.455
C08652=1234.972,102.083,-47.458,-178.346,5.467,148.456
C08653=1234.978,101.834,-47.440,-178.348,5.466,148.456
C08654=1234.982,101.584,-47.421,-178.350,5.465,148.457
C08655=1234.987,101.336,-47.402,-178.353,5.465,148.458
C08656=1234.992,101.086,-47.383,-178.356,5.463,148.458
C08657=1234.997,100.837,-47.364,-178.359,5.462,148.459
C08658=1235.001,100.588,-47.345,-178.361,5.461,148.459
C08659=1235.007,100.338,-47.326,-178.363,5.461,148.460
C08660=1235.011,100.089,-47.307,-178.366,5.460,148.461
C08661=1235.016,99.840,-47.288,-178.368,5.459,148.461
C08662=1235.021,99.591,-47.270,-178.371,5.459,148.462
C08663=1235.026,99.341,-47.250,-178.373,5.458,148.462
C08664=1235.030,99.092,-47.232,-178.376,5.457,148.463
C08665=1235.034,98.843,-47.213,-178.379,5.456,148.463
C08666=1235.040,98.593,-47.195,-178.381,5.455,148.464
C08667=1235.045,98.345,-47.176,-178.384,5.454,148.465
C08668=1235.049,98.095,-47.156,-178.387,5.454,148.465
C08669=1235.054,97.846,-47.138,-178.389,5.453,148.466
C08670=1235.059,97.596,-47.119,-178.391,5.452,148.466
C08671=1235.064,97.347,-47.101,-178.394,5.452,148.467
C08672=1235.069,97.099,-47.082,-178.396,5.451,148.467
C08673=1235.074,96.848,-47.063,-178.399,5.450,148.468
C08674=1235.078,96.600,-47.044,-178.401,5.449,148.469
C08675=1235.083,96.350,-47.025,-178.405,5.448,148.469
C08676=1235.088,96.101,-47.007,-178.407,5.447,148.470
C08677=1235.093,95.852,-46.989,-178.409,5.446,148.470
C08678=1235.098,95.602,-46.969,-178.412,5.446,148.471
C08679=1235.103,95.353,-46.951,-178.414,5.445,148.472
C08680=1235.108,95.104,-46.932,-178.417,5.444,148.472
C08681=1235.112,94.854,-46.914,-178.419,5.444,148.473
C08682=1235.117,94.606,-46.895,-178.422,5.443,148.473
C08683=1235.122,94.356,-46.876,-178.424,5.442,148.474
C08684=1235.127,94.107,-46.858,-178.427,5.441,148.474
C08685=1235.131,93.858,-46.839,-178.429,5.441,148.475
C08686=1235.137,93.609,-46.821,-178.432,5.440,148.476
C08687=1235.141,93.359,-46.802,-178.435,5.439,148.476
C08688=1235.146,93.110,-46.784,-178.437,5.438,148.477
C08689=1235.152,92.861,-46.765,-178.440,5.437,148.477
C08690=1235.156,92.611,-46.746,-178.442,5.437,148.478
C08691=1235.160,92.362,-46.728,-178.445,5.436,148.479
C08692=1235.165,92.113,-46.710,-178.447,5.435,148.479
C08693=1235.170,91.863,-46.690,-178.450,5.434,148.480
C08694=1235.175,91.614,-46.672,-178.452,5.434,148.480
C08695=1235.180,91.365,-46.654,-178.455,5.433,148.481
C08696=1235.184,91.116,-46.635,-178.457,5.432,148.482
C08697=1235.190,90.866,-46.617,-178.460,5.432,148.482
C08698=1235.195,90.617,-46.599,-178.462,5.431,148.483
C08699=1235.199,90.369,-46.580,-178.465,5.430,148.484
C08700=1235.203,90.119,-46.562,-178.468,5.430,148.484
C08701=1235.209,89.869,-46.543,-178.470,5.428,148.485
C08702=1235.214,89.620,-46.525,-178.473,5.427,148.485
C08703=1235.219,89.372,-46.506,-178.476,5.427,148.486
C08704=1235.223,89.122,-46.488,-178.478,5.426,148.487
C08705=1235.229,88.872,-46.470,-178.480,5.425,148.487
C08706=1235.234,88.623,-46.452,-178.483,5.425,148.488
C08707=1235.238,88.374,-46.433,-178.486,5.424,148.488
C08708=1235.242,88.125,-46.415,-178.488,5.423,148.489
C08709=1235.247,87.875,-46.397,-178.490,5.422,148.489
C08710=1235.253,87.626,-46.378,-178.493,5.422,148.490
C08711=1235.258,87.377,-46.360,-178.496,5.421,148.491
C08712=1235.262,87.127,-46.341,-178.498,5.420,148.491
C08713=1235.267,86.878,-46.323,-178.501,5.420,148.492
C08714=1235.272,86.629,-46.305,-178.503,5.419,148.492
C08715=1235.277,86.380,-46.287,-178.506,5.418,148.493
C08716=1235.282,86.130,-46.268,-178.508,5.418,148.494
C08717=1235.287,85.881,-46.250,-178.511,5.417,148.494
C08718=1235.292,85.631,-46.232,-178.513,5.416,148.495
C08719=1235.296,85.383,-46.213,-178.516,5.416,148.495
C08720=1235.301,85.134,-46.195,-178.518,5.415,148.496
C08721=1235.305,84.884,-46.177,-178.521,5.414,148.497
C08722=1235.310,84.635,-46.159,-178.523,5.414,148.497
C08723=1235.315,84.385,-46.141,-178.526,5.412,148.498
C08724=1235.320,84.136,-46.123,-178.529,5.411,148.498
C08725=1235.326,83.887,-46.105,-178.531,5.411,148.499
C08726=1235.330,83.637,-46.086,-178.534,5.410,148.500
C08727=1235.335,83.388,-46.068,-178.537,5.410,148.500
C08728=1235.340,83.139,-46.050,-178.539,5.409,148.501
C08729=1235.345,82.889,-46.032,-178.541,5.408,148.502
C08730=1235.350,82.640,-46.014,-178.544,5.407,148.502
C08731=1235.355,82.391,-45.996,-178.547,5.407,148.503
C08732=1235.360,82.123,-45.977,-178.549,5.406,148.503
C08733=1235.365,81.854,-45.957,-178.552,5.406,148.504
C08734=1235.370,81.586,-45.938,-178.554,5.405,148.505
C08735=1235.376,81.318,-45.918,-178.557,5.404,148.505
C08736=1235.380,81.068,-45.900,-178.560,5.404,148.506
C08737=1235.385,80.819,-45.882,-178.562,5.403,148.507
C08738=1235.390,80.569,-45.864,-178.564,5.402,148.507
C08739=1235.395,80.320,-45.846,-178.568,5.401,148.508
C08740=1235.400,80.070,-45.829,-178.570,5.400,148.508
C08741=1235.405,79.821,-45.811,-178.573,5.400,148.509
C08742=1235.410,79.572,-45.793,-178.576,5.399,148.510
C08743=1235.415,79.323,-45.775,-178.578,5.398,148.510
C08744=1235.419,79.073,-45.756,-178.580,5.397,148.511
C08745=1235.424,78.824,-45.738,-178.583,5.397,148.512
C08746=1235.429,78.575,-45.720,-178.586,5.396,148.512
C08747=1235.434,78.326,-45.702,-178.588,5.396,148.513
C08748=1235.438,78.077,-45.685,-178.590,5.395,148.513
C08749=1235.443,77.827,-45.668,-178.593,5.394,148.514
C08750=1235.448,77.578,-45.650,-178.596,5.393,148.515
C08751=1235.453,77.329,-45.632,-178.598,5.393,148.515
C08752=1235.458,77.079,-45.614,-178.601,5.392,148.516
C08753=1235.463,76.830,-45.596,-178.603,5.392,148.517
C08754=1235.468,76.581,-45.578,-178.606,5.391,148.517
C08755=1235.472,76.330,-45.560,-178.608,5.390,148.518
C08756=1235.477,76.081,-45.542,-178.611,5.389,148.518
C08757=1235.482,75.832,-45.524,-178.613,5.389,148.519
C08758=1235.487,75.583,-45.506,-178.616,5.388,148.520
C08759=1235.492,75.334,-45.488,-178.619,5.388,148.520
C08760=1235.496,75.084,-45.472,-178.621,5.387,148.521
C08761=1235.501,74.835,-45.454,-178.623,5.386,148.521
C08762=1235.506,74.586,-45.436,-178.626,5.386,148.522
C08763=1235.511,74.337,-45.418,-178.628,5.386,148.523
C08764=1235.516,74.087,-45.400,-178.631,5.385,148.523
C08765=1235.521,73.838,-45.382,-178.633,5.385,148.524
C08766=1235.526,73.589,-45.364,-178.636,5.384,148.524
C08767=1235.531,73.339,-45.348,-178.638,5.383,148.525
C08768=1235.536,73.090,-45.330,-178.641,5.382,148.526
C08769=1235.540,72.841,-45.312,-178.643,5.382,148.526
C08770=1235.546,72.591,-45.294,-178.646,5.381,148.527
C08771=1235.551,72.342,-45.276,-178.649,5.381,148.528
C08772=1235.556,72.093,-45.259,-178.651,5.380,148.528
C08773=1235.560,71.843,-45.242,-178.653,5.379,148.529
C08774=1235.565,71.594,-45.224,-178.656,5.378,148.530
C08775=1235.570,71.345,-45.206,-178.659,5.378,148.530
C08776=1235.575,71.095,-45.189,-178.661,5.377,148.531
C08777=1235.580,70.846,-45.171,-178.664,5.377,148.532
C08778=1235.584,70.597,-45.153,-178.666,5.376,148.532
C08779=1235.589,70.347,-45.136,-178.669,5.375,148.533
C08780=1235.594,70.098,-45.118,-178.671,5.375,148.533
C08781=1235.599,69.848,-45.101,-178.674,5.374,148.534
C08782=1235.604,69.599,-45.083,-178.677,5.373,148.535
C08783=1235.609,69.350,-45.066,-178.679,5.373,148.535
C08784=1235.614,69.100,-45.048,-178.682,5.372,148.536
C08785=1235.619,68.851,-45.030,-178.684,5.371,148.536
C08786=1235.623,68.602,-45.013,-178.687,5.371,148.537
C08787=1235.628,68.353,-44.995,-178.689,5.370,148.538
C08788=1235.633,68.103,-44.978,-178.692,5.369,148.538
C08789=1235.637,67.854,-44.961,-178.695,5.369,148.539
C08790=1235.643,67.604,-44.944,-178.697,5.368,148.540
C08791=1235.648,67.356,-44.926,-178.700,5.368,148.540
C08792=1235.653,67.106,-44.909,-178.702,5.367,148.541
C08793=1235.658,66.857,-44.891,-178.704,5.367,148.541
C08794=1235.663,66.607,-44.874,-178.707,5.366,148.542
C08795=1235.668,66.358,-44.856,-178.709,5.366,148.543
C08796=1235.672,66.108,-44.839,-178.712,5.365,148.543
C08797=1235.677,65.859,-44.821,-178.715,5.365,148.544
C08798=1235.682,65.610,-44.805,-178.717,5.364,148.545
C08799=1235.687,65.360,-44.787,-178.720,5.363,148.545
C08800=1235.692,65.111,-44.770,-178.722,5.362,148.546
C08801=1235.696,64.861,-44.753,-178.725,5.362,148.547
C08802=1235.702,64.613,-44.735,-178.727,5.361,148.547
C08803=1235.707,64.363,-44.718,-178.730,5.361,148.548
C08804=1235.711,64.114,-44.701,-178.732,5.360,148.548
C08805=1235.716,63.864,-44.683,-178.735,5.360,148.549
C08806=1235.722,63.615,-44.666,-178.738,5.359,148.550
C08807=1235.726,63.366,-44.649,-178.740,5.358,148.550
C08808=1235.731,63.116,-44.631,-178.742,5.357,148.551
C08809=1235.735,62.867,-44.615,-178.745,5.357,148.552
C08810=1235.741,62.618,-44.597,-178.747,5.357,148.552
C08811=1235.746,62.368,-44.580,-178.750,5.356,148.553
C08812=1235.751,62.119,-44.563,-178.752,5.356,148.554
C08813=1235.756,61.870,-44.545,-178.755,5.355,148.554
C08814=1235.760,61.620,-44.529,-178.758,5.355,148.555
C08815=1235.765,61.370,-44.511,-178.760,5.354,148.556
C08816=1235.770,61.121,-44.495,-178.762,5.353,148.556
C08817=1235.775,60.872,-44.477,-178.765,5.353,148.557
C08818=1235.780,60.623,-44.460,-178.768,5.352,148.557
C08819=1235.785,60.373,-44.443,-178.770,5.351,148.558
C08820=1235.789,60.124,-44.426,-178.773,5.351,148.559
C08821=1235.794,59.874,-44.408,-178.776,5.350,148.559
C08822=1235.800,59.625,-44.391,-178.778,5.350,148.560
C08823=1235.805,59.376,-44.375,-178.780,5.350,148.561
C08824=1235.810,59.126,-44.358,-178.783,5.349,148.561
C08825=1235.814,58.877,-44.340,-178.785,5.348,148.562
C08826=1235.819,58.627,-44.323,-178.788,5.348,148.562
C08827=1235.824,58.378,-44.306,-178.790,5.347,148.563
C08828=1235.830,58.129,-44.289,-178.793,5.347,148.564
C08829=1235.834,57.879,-44.273,-178.796,5.346,148.564
C08830=1235.838,57.630,-44.255,-178.798,5.345,148.565
C08831=1235.843,57.381,-44.238,-178.801,5.345,148.566
C08832=1235.848,57.132,-44.222,-178.804,5.344,148.566
C08833=1235.854,56.882,-44.204,-178.806,5.344,148.567
C08834=1235.858,56.633,-44.188,-178.808,5.344,148.568
C08835=1235.863,56.383,-44.171,-178.810,5.343,148.568
C08836=1235.869,56.115,-44.153,-178.814,5.343,148.569
C08837=1235.874,55.846,-44.134,-178.816,5.342,148.570
C08838=1235.879,55.578,-44.116,-178.819,5.342,148.570
C08839=1235.885,55.309,-44.098,-178.822,5.340,148.571
C08840=1235.889,55.060,-44.081,-178.824,5.340,148.572
C08841=1235.895,54.811,-44.064,-178.827,5.340,148.572
C08842=1235.899,54.561,-44.047,-178.829,5.339,148.573
C08843=1235.904,54.312,-44.030,-178.832,5.339,148.574
C08844=1235.909,54.063,-44.013,-178.835,5.338,148.574
C08845=1235.914,53.814,-43.996,-178.837,5.337,148.575
C08846=1235.919,53.564,-43.979,-178.839,5.337,148.576
C08847=1235.924,53.315,-43.963,-178.842,5.336,148.576
C08848=1235.928,53.065,-43.946,-178.845,5.335,148.577
C08849=1235.934,52.816,-43.929,-178.847,5.336,148.578
C08850=1235.938,52.566,-43.912,-178.849,5.335,148.578
C08851=1235.943,52.317,-43.896,-178.852,5.334,148.579
C08852=1235.949,52.068,-43.879,-178.855,5.334,148.580
C08853=1235.953,51.818,-43.862,-178.857,5.333,148.580
C08854=1235.958,51.569,-43.845,-178.860,5.333,148.581
C08855=1235.963,51.320,-43.829,-178.863,5.332,148.582
C08856=1235.968,51.070,-43.812,-178.865,5.332,148.582
C08857=1235.972,50.821,-43.795,-178.867,5.331,148.583
C08858=1235.978,50.570,-43.779,-178.869,5.331,148.583
C08859=1235.983,50.322,-43.762,-178.872,5.330,148.584
C08860=1235.988,50.072,-43.746,-178.875,5.330,148.585
C08861=1235.992,49.823,-43.729,-178.877,5.329,148.585
C08862=1235.998,49.574,-43.712,-178.880,5.329,148.586
C08863=1236.002,49.324,-43.695,-178.883,5.328,148.587
C08864=1236.007,49.075,-43.679,-178.885,5.327,148.587
C08865=1236.013,48.826,-43.662,-178.887,5.328,148.588
C08866=1236.017,48.576,-43.645,-178.890,5.327,148.589
C08867=1236.022,48.327,-43.629,-178.893,5.327,148.589
C08868=1236.027,48.077,-43.613,-178.895,5.326,148.590
C08869=1236.032,47.827,-43.596,-178.898,5.325,148.591
C08870=1236.037,47.579,-43.579,-178.900,5.325,148.591
C08871=1236.042,47.329,-43.563,-178.903,5.324,148.592
C08872=1236.046,47.080,-43.546,-178.905,5.323,148.593
C08873=1236.052,46.831,-43.529,-178.907,5.324,148.593
C08874=1236.057,46.580,-43.513,-178.910,5.323,148.594
C08875=1236.061,46.331,-43.496,-178.913,5.322,148.595
C08876=1236.066,46.082,-43.480,-178.915,5.322,148.595
C08877=1236.071,45.833,-43.464,-178.918,5.321,148.596
C08878=1236.077,45.584,-43.447,-178.920,5.321,148.597
C08879=1236.081,45.333,-43.431,-178.923,5.320,148.597
C08880=1236.086,45.084,-43.414,-178.925,5.320,148.598
C08881=1236.091,44.835,-43.398,-178.928,5.320,148.599
C08882=1236.096,44.586,-43.381,-178.930,5.319,148.599
C08883=1236.101,44.336,-43.365,-178.933,5.319,148.600
C08884=1236.106,44.087,-43.348,-178.936,5.318,148.601
C08885=1236.111,43.837,-43.332,-178.938,5.317,148.601
C08886=1236.116,43.588,-43.316,-178.940,5.318,148.602
C08887=1236.120,43.338,-43.299,-178.943,5.317,148.602
C08888=1236.126,43.089,-43.283,-178.945,5.316,148.603
C08889=1236.130,42.840,-43.266,-178.948,5.316,148.604
C08890=1236.135,42.591,-43.251,-178.951,5.315,148.604
C08891=1236.141,42.341,-43.233,-178.953,5.314,148.605
C08892=1236.145,42.091,-43.217,-178.956,5.314,148.606
C08893=1236.151,41.842,-43.201,-178.958,5.314,148.606
C08894=1236.155,41.592,-43.184,-178.961,5.314,148.607
C08895=1236.160,41.344,-43.168,-178.963,5.313,148.608
C08896=1236.165,41.093,-43.152,-178.966,5.312,148.608
C08897=1236.170,40.845,-43.136,-178.968,5.312,148.609
C08898=1236.175,40.595,-43.120,-178.971,5.311,148.610
C08899=1236.180,40.346,-43.104,-178.973,5.312,148.611
C08900=1236.184,40.096,-43.087,-178.976,5.311,148.611
C08901=1236.190,39.847,-43.071,-178.978,5.310,148.612
C08902=1236.195,39.597,-43.054,-178.981,5.310,148.613
C08903=1236.200,39.348,-43.039,-178.984,5.309,148.613
C08904=1236.205,39.098,-43.022,-178.986,5.309,148.614
C08905=1236.210,38.849,-43.006,-178.988,5.309,148.615
C08906=1236.215,38.599,-42.990,-178.991,5.308,148.615
C08907=1236.220,38.351,-42.973,-178.994,5.308,148.616
C08908=1236.224,38.100,-42.957,-178.996,5.307,148.617
C08909=1236.230,37.852,-42.941,-178.999,5.307,148.617
C08910=1236.234,37.602,-42.925,-179.001,5.306,148.618
C08911=1236.239,37.353,-42.909,-179.003,5.306,148.618
C08912=1236.244,37.103,-42.893,-179.006,5.305,148.619
C08913=1236.249,36.854,-42.877,-179.008,5.305,148.620
C08914=1236.254,36.604,-42.861,-179.011,5.304,148.620
C08915=1236.259,36.355,-42.844,-179.014,5.304,148.621
C08916=1236.264,36.105,-42.828,-179.016,5.304,148.622
C08917=1236.269,35.855,-42.813,-179.018,5.303,148.622
C08918=1236.274,35.606,-42.796,-179.021,5.303,148.623
C08919=1236.279,35.357,-42.781,-179.024,5.302,148.624
C08920=1236.284,35.108,-42.764,-179.026,5.302,148.624
C08921=1236.289,34.858,-42.748,-179.029,5.301,148.625
C08922=1236.294,34.609,-42.732,-179.031,5.301,148.626
C08923=1236.299,34.359,-42.716,-179.034,5.301,148.627
C08924=1236.303,34.110,-42.700,-179.036,5.300,148.627
C08925=1236.308,33.860,-42.684,-179.039,5.300,148.628
C08926=1236.313,33.611,-42.669,-179.042,5.299,148.629
C08927=1236.318,33.361,-42.652,-179.044,5.299,148.629
C08928=1236.323,33.112,-42.636,-179.046,5.299,148.630
C08929=1236.329,32.863,-42.621,-179.049,5.298,148.631
C08930=1236.333,32.613,-42.604,-179.052,5.298,148.631
C08931=1236.339,32.364,-42.589,-179.054,5.297,148.632
C08932=1236.343,32.114,-42.573,-179.056,5.297,148.633
C08933=1236.348,31.865,-42.556,-179.059,5.297,148.633
C08934=1236.353,31.616,-42.541,-179.062,5.296,148.634
C08935=1236.358,31.366,-42.525,-179.064,5.296,148.635
C08936=1236.363,31.117,-42.509,-179.067,5.295,148.635
C08937=1236.368,30.867,-42.493,-179.069,5.295,148.636
C08938=1236.373,30.617,-42.478,-179.072,5.295,148.637
C08939=1236.378,30.369,-42.461,-179.074,5.294,148.637
C08940=1236.383,30.099,-42.444,-179.077,5.294,148.638
C08941=1236.389,29.831,-42.427,-179.080,5.293,148.639
C08942=1236.394,29.563,-42.410,-179.082,5.293,148.639
C08943=1236.399,29.294,-42.393,-179.085,5.292,148.640
C08944=1236.404,29.044,-42.377,-179.087,5.293,148.641
C08945=1236.409,28.795,-42.362,-179.090,5.292,148.642
C08946=1236.415,28.545,-42.346,-179.093,5.292,148.642
C08947=1236.419,28.296,-42.330,-179.095,5.291,148.643
C08948=1236.424,28.047,-42.315,-179.098,5.290,148.644
C08949=1236.429,27.797,-42.299,-179.100,5.291,148.644
C08950=1236.434,27.547,-42.283,-179.103,5.290,148.645
C08951=1236.439,27.298,-42.268,-179.105,5.290,148.646
C08952=1236.444,27.049,-42.251,-179.108,5.289,148.646
C08953=1236.448,26.799,-42.236,-179.111,5.288,148.647
C08954=1236.454,26.550,-42.220,-179.113,5.289,148.648
C08955=1236.459,26.300,-42.205,-179.115,5.288,148.648
C08956=1236.464,26.050,-42.189,-179.118,5.287,148.649
C08957=1236.469,25.801,-42.174,-179.120,5.287,148.650
C08958=1236.474,25.552,-42.158,-179.122,5.287,148.650
C08959=1236.479,25.302,-42.141,-179.125,5.286,148.651
C08960=1236.484,25.053,-42.126,-179.128,5.286,148.652
C08961=1236.489,24.804,-42.111,-179.130,5.285,148.652
C08962=1236.493,24.554,-42.095,-179.133,5.285,148.653
C08963=1236.499,24.304,-42.079,-179.135,5.285,148.654
C08964=1236.503,24.055,-42.064,-179.138,5.284,148.654
C08965=1236.509,23.806,-42.049,-179.140,5.284,148.655
C08966=1236.514,23.556,-42.033,-179.143,5.283,148.656
C08967=1236.518,23.307,-42.018,-179.145,5.284,148.656
C08968=1236.524,23.057,-42.002,-179.148,5.283,148.657
C08969=1236.528,22.807,-41.986,-179.150,5.282,148.658
C08970=1236.534,22.558,-41.971,-179.153,5.282,148.658
C08971=1236.538,22.309,-41.956,-179.155,5.283,148.659
C08972=1236.544,22.059,-41.940,-179.158,5.282,148.660
C08973=1236.549,21.809,-41.924,-179.161,5.281,148.661
C08974=1236.553,21.560,-41.909,-179.163,5.281,148.661
C08975=1236.559,21.311,-41.894,-179.165,5.281,148.662
C08976=1236.563,21.062,-41.879,-179.168,5.281,148.663
C08977=1236.568,20.811,-41.863,-179.171,5.280,148.663
C08978=1236.573,20.562,-41.847,-179.173,5.279,148.664
C08979=1236.578,20.313,-41.832,-179.176,5.279,148.665
C08980=1236.584,20.064,-41.816,-179.178,5.279,148.666
C08981=1236.588,19.813,-41.801,-179.181,5.279,148.666
C08982=1236.593,19.564,-41.786,-179.183,5.278,148.667
C08983=1236.598,19.315,-41.770,-179.186,5.278,148.668
C08984=1236.603,19.066,-41.755,-179.188,5.278,148.668
C08985=1236.608,18.816,-41.739,-179.191,5.277,148.669
C08986=1236.613,18.566,-41.723,-179.193,5.277,148.670
C08987=1236.618,18.317,-41.708,-179.196,5.276,148.670
C08988=1236.623,18.068,-41.693,-179.198,5.276,148.671
C08989=1236.628,17.819,-41.678,-179.201,5.276,148.672
C08990=1236.634,17.569,-41.663,-179.203,5.275,148.672
C08991=1236.638,17.319,-41.648,-179.206,5.275,148.673
C08992=1236.643,17.070,-41.632,-179.208,5.275,148.674
C08993=1236.648,16.820,-41.616,-179.211,5.274,148.674
C08994=1236.653,16.571,-41.601,-179.213,5.274,148.675
C08995=1236.658,16.322,-41.586,-179.216,5.274,148.676
C08996=1236.662,16.072,-41.570,-179.218,5.274,148.676
C08997=1236.668,15.822,-41.556,-179.221,5.273,148.677
C08998=1236.673,15.573,-41.541,-179.224,5.273,148.678
C08999=1236.678,15.323,-41.525,-179.226,5.273,148.678
C09000=1236.683,15.074,-41.510,-179.228,5.272,148.679
C09001=1236.688,14.825,-41.494,-179.231,5.272,148.680
C09002=1236.693,14.574,-41.480,-179.234,5.271,148.681
C09003=1236.698,14.325,-41.464,-179.236,5.271,148.681
C09004=1236.703,14.076,-41.449,-179.238,5.271,148.682
C09005=1236.708,13.827,-41.434,-179.241,5.270,148.683
C09006=1236.713,13.577,-41.419,-179.244,5.270,148.683
C09007=1236.718,13.327,-41.404,-179.246,5.270,148.684
C09008=1236.723,13.078,-41.389,-179.248,5.270,148.685
C09009=1236.728,12.828,-41.373,-179.251,5.269,148.685
C09010=1236.733,12.579,-41.359,-179.253,5.269,148.686
C09011=1236.738,12.329,-41.343,-179.256,5.269,148.687
C09012=1236.743,12.080,-41.328,-179.258,5.268,148.687
C09013=1236.747,11.831,-41.313,-179.261,5.268,148.688
C09014=1236.753,11.581,-41.298,-179.263,5.268,148.689
C09015=1236.758,11.332,-41.283,-179.266,5.267,148.689
C09016=1236.763,11.082,-41.268,-179.268,5.267,148.690
C09017=1236.768,10.833,-41.253,-179.271,5.266,148.691
C09018=1236.773,10.583,-41.237,-179.273,5.267,148.692
C09019=1236.778,10.334,-41.222,-179.276,5.266,148.692
C09020=1236.782,10.084,-41.208,-179.278,5.265,148.693
C09021=1236.788,9.834,-41.192,-179.280,5.266,148.694
C09022=1236.792,9.585,-41.177,-179.283,5.265,148.694
C09023=1236.797,9.336,-41.163,-179.286,5.265,148.695
C09024=1236.803,9.086,-41.148,-179.289,5.264,148.696
C09025=1236.808,8.837,-41.133,-179.291,5.265,148.697
C09026=1236.813,8.587,-41.118,-179.294,5.264,148.697
C09027=1236.818,8.338,-41.103,-179.296,5.264,148.698
C09028=1236.823,8.088,-41.088,-179.298,5.264,148.699
C09029=1236.828,7.839,-41.073,-179.301,5.263,148.699
C09030=1236.833,7.589,-41.059,-179.304,5.263,148.700
C09031=1236.838,7.340,-41.044,-179.306,5.262,148.701
C09032=1236.843,7.089,-41.028,-179.308,5.263,148.701
C09033=1236.848,6.840,-41.013,-179.311,5.262,148.702
C09034=1236.852,6.591,-40.999,-179.314,5.261,148.703
C09035=1236.858,6.341,-40.984,-179.316,5.262,148.703
C09036=1236.863,6.092,-40.969,-179.318,5.261,148.704
C09037=1236.867,5.842,-40.954,-179.321,5.261,148.705
C09038=1236.873,5.593,-40.939,-179.324,5.260,148.705
C09039=1236.878,5.343,-40.924,-179.326,5.260,148.706
C09040=1236.882,5.094,-40.909,-179.328,5.260,148.707
C09041=1236.887,4.844,-40.895,-179.331,5.259,148.708
C09042=1236.893,4.595,-40.880,-179.333,5.260,148.708
C09043=1236.898,4.345,-40.865,-179.336,5.259,148.709
C09044=1236.903,4.077,-40.850,-179.339,5.259,148.710
C09045=1236.909,3.807,-40.833,-179.342,5.258,148.711
C09046=1236.914,3.539,-40.818,-179.344,5.258,148.711
C09047=1236.919,3.270,-40.802,-179.346,5.258,148.712
C09048=1236.925,3.020,-40.787,-179.349,5.258,148.713
C09049=1236.929,2.771,-40.772,-179.352,5.257,148.714
C09050=1236.934,2.521,-40.758,-179.354,5.258,148.714
C09051=1236.939,2.272,-40.743,-179.357,5.257,148.715
C09052=1236.945,2.022,-40.728,-179.360,5.257,148.716
C09053=1236.950,1.772,-40.714,-179.362,5.256,148.716
C09054=1236.954,1.523,-40.699,-179.364,5.256,148.717
C09055=1236.960,1.274,-40.685,-179.367,5.256,148.718
C09056=1236.964,1.025,-40.670,-179.370,5.255,148.718
C09057=1236.970,0.775,-40.655,-179.372,5.256,148.719
C09058=1236.975,0.525,-40.640,-179.374,5.255,148.720
C09059=1236.980,0.276,-40.625,-179.377,5.254,148.720
C09060=1236.985,0.027,-40.611,-179.379,5.255,148.721
C09061=1236.990,-0.223,-40.597,-179.382,5.254,148.722
C09062=1236.994,-0.472,-40.582,-179.384,5.254,148.722
C09063=1237.000,-0.722,-40.567,-179.386,5.254,148.723
C09064=1237.005,-0.972,-40.553,-179.389,5.253,148.724
C09065=1237.010,-1.221,-40.538,-179.392,5.253,148.725
C09066=1237.015,-1.471,-40.524,-179.394,5.253,148.725
C09067=1237.020,-1.721,-40.509,-179.396,5.253,148.726
C09068=1237.024,-1.970,-40.495,-179.399,5.252,148.727
C09069=1237.030,-2.220,-40.479,-179.401,5.252,148.727
C09070=1237.035,-2.469,-40.465,-179.404,5.252,148.728
C09071=1237.040,-2.718,-40.451,-179.407,5.252,148.729
C09072=1237.045,-2.968,-40.437,-179.409,5.252,148.730
C09073=1237.050,-3.217,-40.422,-179.412,5.251,148.730
C09074=1237.055,-3.467,-40.408,-179.414,5.251,148.731
C09075=1237.060,-3.717,-40.393,-179.417,5.250,148.732
C09076=1237.065,-3.966,-40.379,-179.419,5.251,148.732
C09077=1237.069,-4.215,-40.364,-179.422,5.250,148.733
C09078=1237.074,-4.465,-40.350,-179.424,5.250,148.734
C09079=1237.080,-4.715,-40.335,-179.426,5.250,148.734
C09080=1237.086,-4.964,-40.321,-179.429,5.249,148.735
C09081=1237.091,-5.214,-40.307,-179.432,5.249,148.736
C09082=1237.096,-5.464,-40.292,-179.434,5.249,148.736
C09083=1237.100,-5.713,-40.277,-179.437,5.249,148.737
C09084=1237.105,-5.962,-40.263,-179.439,5.248,148.738
C09085=1237.110,-6.212,-40.249,-179.441,5.248,148.739
C09086=1237.115,-6.462,-40.235,-179.444,5.248,148.739
C09087=1237.120,-6.711,-40.220,-179.447,5.248,148.740
C09088=1237.126,-6.960,-40.206,-179.449,5.248,148.741
C09089=1237.131,-7.210,-40.192,-179.452,5.247,148.742
C09090=1237.135,-7.459,-40.177,-179.454,5.247,148.742
C09091=1237.140,-7.709,-40.163,-179.457,5.247,148.743
C09092=1237.145,-7.959,-40.149,-179.459,5.247,148.744
C09093=1237.150,-8.208,-40.134,-179.461,5.247,148.744
C09094=1237.156,-8.457,-40.120,-179.464,5.246,148.745
C09095=1237.161,-8.707,-40.106,-179.467,5.246,148.746
C09096=1237.166,-8.957,-40.092,-179.469,5.246,148.746
C09097=1237.170,-9.207,-40.078,-179.471,5.246,148.747
C09098=1237.175,-9.456,-40.063,-179.474,5.245,148.748
C09099=1237.181,-9.705,-40.049,-179.476,5.245,148.748
C09100=1237.186,-9.955,-40.035,-179.479,5.245,148.749
C09101=1237.191,-10.205,-40.021,-179.481,5.244,148.750
C09102=1237.196,-10.454,-40.007,-179.483,5.245,148.751
C09103=1237.201,-10.704,-39.992,-179.487,5.244,148.751
C09104=1237.206,-10.954,-39.978,-179.489,5.244,148.752
C09105=1237.211,-11.203,-39.964,-179.491,5.244,148.753
C09106=1237.216,-11.453,-39.950,-179.494,5.244,148.754
C09107=1237.221,-11.702,-39.936,-179.497,5.243,148.754
C09108=1237.225,-11.952,-39.922,-179.499,5.243,148.755
C09109=1237.231,-12.201,-39.908,-179.501,5.243,148.756
C09110=1237.236,-12.450,-39.894,-179.504,5.242,148.756
C09111=1237.241,-12.700,-39.879,-179.506,5.243,148.757
C09112=1237.246,-12.950,-39.865,-179.509,5.242,148.758
C09113=1237.251,-13.199,-39.851,-179.511,5.242,148.758
C09114=1237.256,-13.449,-39.837,-179.514,5.242,148.759
C09115=1237.261,-13.698,-39.823,-179.516,5.241,148.760
C09116=1237.266,-13.948,-39.808,-179.518,5.242,148.761
C09117=1237.271,-14.197,-39.795,-179.521,5.241,148.761
C09118=1237.276,-14.447,-39.782,-179.524,5.241,148.762
C09119=1237.281,-14.697,-39.767,-179.526,5.241,148.763
C09120=1237.286,-14.946,-39.753,-179.529,5.241,148.764
C09121=1237.292,-15.195,-39.739,-179.531,5.240,148.764
C09122=1237.297,-15.445,-39.725,-179.534,5.241,148.765
C09123=1237.302,-15.695,-39.711,-179.536,5.240,148.766
C09124=1237.306,-15.944,-39.697,-179.539,5.239,148.766
C09125=1237.312,-16.193,-39.683,-179.541,5.240,148.767
C09126=1237.317,-16.444,-39.669,-179.544,5.239,148.768
C09127=1237.322,-16.693,-39.655,-179.546,5.240,148.768
C09128=1237.327,-16.942,-39.641,-179.548,5.239,148.769
C09129=1237.332,-17.192,-39.627,-179.551,5.239,148.770
C09130=1237.336,-17.441,-39.613,-179.553,5.239,148.770
C09131=1237.342,-17.692,-39.600,-179.556,5.238,148.771
C09132=1237.347,-17.941,-39.586,-179.558,5.238,148.772
C09133=1237.352,-18.190,-39.571,-179.561,5.238,148.773
